LIN {X 0,Y 551.057,Z 884.33,A -85,B 0,C 180,E1 23176.84,E2 23176.84} C_VEL
LIN {X 0,Y 547.83,Z 907.139,A -85,B 0,C 180,E1 23175.833,E2 23175.833} C_VEL
LIN {X 0,Y 543.815,Z 933.396,A -85,B 0,C 180,E1 23174.47,E2 23174.47} C_VEL
LIN {X 0,Y 539.915,Z 957.037,A -85,B 0,C 180,E1 23173.041,E2 23173.041} C_VEL
LIN {X 0,Y 534.4,Z 990.703,A -85,B 0,C 180,E1 23170.731,E2 23170.731} C_VEL
LIN {X 0,Y 530.47,Z 1014.088,A -85,B 0,C 180,E1 23168.879,E2 23168.879} C_VEL
LIN {X 0,Y 527.355,Z 1031.726,A -85,B 0,C 180,E1 23167.286,E2 23167.286} C_VEL
LIN {X 0,Y 524.138,Z 1048.925,A -85,B 0,C 180,E1 23165.514,E2 23165.514} C_VEL
LIN {X 0,Y 520.353,Z 1068.496,A -85,B 0,C 180,E1 23163.207,E2 23163.207} C_VEL
LIN {X 0,Y 517.554,Z 1082.457,A -85,B 0,C 180,E1 23161.313,E2 23161.313} C_VEL
LIN {X 0,Y 514.336,Z 1098.584,A -85,B 0,C 180,E1 23158.825,E2 23158.825} C_VEL
LIN {X 0,Y 511.848,Z 1111.312,A -85,B 0,C 180,E1 23156.53,E2 23156.53} C_VEL
LIN {X 0,Y 509.597,Z 1122.961,A -85,B 0,C 180,E1 23154.088,E2 23154.088} C_VEL
LIN {X 0,Y 507.873,Z 1132.943,A -85,B 0,C 180,E1 23151.725,E2 23151.725} C_VEL
LIN {X 0,Y 506.606,Z 1141.31,A -85,B 0,C 180,E1 23149.486,E2 23149.486} C_VEL
LIN {X 0,Y 505.604,Z 1149.002,A -85,B 0,C 180,E1 23147.139,E2 23147.139} C_VEL
LIN {X 0,Y 504.896,Z 1155.619,A -85,B 0,C 180,E1 23144.803,E2 23144.803} C_VEL
LIN {X 0,Y 504.42,Z 1161.209,A -85,B 0,C 180,E1 23142.479,E2 23142.479} C_VEL
LIN {X 0,Y 504.14,Z 1166.009,A -85,B 0,C 180,E1 23140.053,E2 23140.053} C_VEL
LIN {X 0,Y 503.99,Z 1169.754,A -85,B 0,C 180,E1 23137.64,E2 23137.64} C_VEL
LIN {X 0,Y 503.929,Z 1172.474,A -85,B 0,C 180,E1 23135.238,E2 23135.238} C_VEL
LIN {X 0,Y 503.908,Z 1174.232,A -85,B 0,C 180,E1 23132.731,E2 23132.731} C_VEL
LIN {X 0,Y 503.897,Z 1174.895,A -85,B 0,C 180,E1 23130.342,E2 23130.342} C_VEL
LIN {X 0,Y 503.911,Z 1174.515,A -85,B 0,C 180,E1 23127.841,E2 23127.841} C_VEL
LIN {X 0,Y 503.919,Z 1173.138,A -85,B 0,C 180,E1 23125.449,E2 23125.449} C_VEL
LIN {X 0,Y 503.964,Z 1170.607,A -85,B 0,C 180,E1 23122.936,E2 23122.936} C_VEL
LIN {X 0,Y 504.088,Z 1167.151,A -85,B 0,C 180,E1 23120.525,E2 23120.525} C_VEL
LIN {X 0,Y 504.351,Z 1162.399,A -85,B 0,C 180,E1 23117.987,E2 23117.987} C_VEL
LIN {X 0,Y 504.788,Z 1156.758,A -85,B 0,C 180,E1 23115.549,E2 23115.549} C_VEL
LIN {X 0,Y 505.495,Z 1149.985,A -85,B 0,C 180,E1 23113.098,E2 23113.098} C_VEL
LIN {X 0,Y 506.451,Z 1142.44,A -85,B 0,C 180,E1 23110.751,E2 23110.751} C_VEL
LIN {X 0,Y 507.667,Z 1134.224,A -85,B 0,C 180,E1 23108.512,E2 23108.512} C_VEL
LIN {X 0,Y 509.239,Z 1124.921,A -85,B 0,C 180,E1 23106.266,E2 23106.266} C_VEL
LIN {X 0,Y 511.074,Z 1115.037,A -85,B 0,C 180,E1 23104.135,E2 23104.135} C_VEL
LIN {X 0,Y 512.89,Z 1105.848,A -85,B 0,C 180,E1 23102.357,E2 23102.357} C_VEL
LIN {X 0,Y 515.553,Z 1092.457,A -85,B 0,C 180,E1 23100.105,E2 23100.105} C_VEL
LIN {X 0,Y 518.946,Z 1075.502,A -85,B 0,C 180,E1 23097.615,E2 23097.615} C_VEL
LIN {X 0,Y 522.004,Z 1059.865,A -85,B 0,C 180,E1 23095.647,E2 23095.647} C_VEL
LIN {X 0,Y 524.918,Z 1044.704,A -85,B 0,C 180,E1 23093.945,E2 23093.945} C_VEL
LIN {X 0,Y 527.865,Z 1028.88,A -85,B 0,C 180,E1 23092.353,E2 23092.353} C_VEL
LIN {X 0,Y 531.711,Z 1007.061,A -85,B 0,C 180,E1 23090.445,E2 23090.445} C_VEL
LIN {X 0,Y 535.099,Z 986.395,A -85,B 0,C 180,E1 23088.874,E2 23088.874} C_VEL
LIN {X 0,Y 540.157,Z 955.538,A -85,B 0,C 180,E1 23086.774,E2 23086.774} C_VEL
LIN {X 0,Y 544.266,Z 930.729,A -85,B 0,C 180,E1 23085.284,E2 23085.284} C_VEL
LIN {X 0,Y 548.137,Z 905.022,A -85,B 0,C 180,E1 23083.979,E2 23083.979} C_VEL
LIN {X 0,Y 551.673,Z 880.009,A -85,B 0,C 180,E1 23082.891,E2 23082.891} C_VEL
LIN {X 0,Y 554.76,Z 854.396,A -85,B 0,C 180,E1 23081.983,E2 23081.983} C_VEL
LIN {X 0,Y 557.091,Z 832.3,A -85,B 0,C 180,E1 23081.336,E2 23081.336} C_VEL
LIN {X 0,Y 559.562,Z 804.066,A -85,B 0,C 180,E1 23080.685,E2 23080.685} C_VEL
LIN {X 0,Y 571.153,Z 655.622,A -85,B 0,C 180,E1 23077.83,E2 23077.83} C_VEL
LIN {X 0,Y 578.577,Z 553.045,A -85,B 0,C 180,E1 23076.025,E2 23076.025} C_VEL
LIN {X 0,Y 583.709,Z 465.889,A -85,B 0,C 180,E1 23074.614,E2 23074.614} C_VEL
LIN {X 0,Y 584.556,Z 445.741,A -85,B 0,C 180,E1 23074.283,E2 23074.283} C_VEL
LIN {X 0,Y 571.093,Z 433.147,A -85,B 0,C 180,E1 23071.921,E2 23071.921} C_VEL
LIN {X 0,Y 562.408,Z 425.648,A -85,B 0,C 180,E1 23070.267,E2 23070.267} C_VEL
LIN {X 0,Y 555.456,Z 419.784,A -85,B 0,C 180,E1 23068.845,E2 23068.845} C_VEL
LIN {X 0,Y 552.715,Z 417.682,A -85,B 0,C 180,E1 23068.24,E2 23068.24} C_VEL
LIN {X 0,Y 551.114,Z 414.287,A -85,B 0,C 180,E1 23066.566,E2 23066.566} C_VEL
LIN {X 0,Y 548.827,Z 409.657,A -85,B 0,C 180,E1 23063.743,E2 23063.743} C_VEL
LIN {X 0,Y 546.381,Z 404.793,A -85,B 0,C 180,E1 23059.221,E2 23059.221} C_VEL
LIN {X 0,Y 545.111,Z 403.52,A -85,B 0,C 180,E1 23054.663,E2 23054.663} C_VEL
LIN {X 0,Y 545.756,Z 404.238,A -85,B 0,C 180,E1 23050.557,E2 23050.557} C_VEL
LIN {X 0,Y 546.687,Z 405.294,A -85,B 0,C 180,E1 23048.52,E2 23048.52} C_VEL
LIN {X 0,Y 549.381,Z 410.452,A -85,B 0,C 180,E1 23044.07,E2 23044.07} C_VEL
LIN {X 0,Y 552.019,Z 415.595,A -85,B 0,C 180,E1 23041.098,E2 23041.098} C_VEL
LIN {X 0,Y 554.609,Z 420.558,A -85,B 0,C 180,E1 23038.76,E2 23038.76} C_VEL
LIN {X 0,Y 557.191,Z 425.708,A -85,B 0,C 180,E1 23036.708,E2 23036.708} C_VEL
LIN {X 0,Y 559.787,Z 430.872,A -85,B 0,C 180,E1 23034.876,E2 23034.876} C_VEL
LIN {X 0,Y 563.507,Z 438.145,A -85,B 0,C 180,E1 23032.557,E2 23032.557} C_VEL
LIN {X 0,Y 567.981,Z 447.698,A -85,B 0,C 180,E1 23029.963,E2 23029.963} C_VEL
LIN {X 0,Y 572.898,Z 458.394,A -85,B 0,C 180,E1 23027.399,E2 23027.399} C_VEL
LIN {X 0,Y 577.116,Z 468.188,A -85,B 0,C 180,E1 23025.322,E2 23025.322} C_VEL
LIN {X 0,Y 570.774,Z 501.691,A -85,B 0,C 180,E1 23022.354,E2 23022.354} C_VEL
LIN {X 0,Y 564.296,Z 538.268,A -85,B 0,C 180,E1 23019.244,E2 23019.244} C_VEL
LIN {X 0,Y 557.893,Z 576.998,A -85,B 0,C 180,E1 23016.066,E2 23016.066} C_VEL
LIN {X 0,Y 553.505,Z 608.409,A -85,B 0,C 180,E1 23013.5,E2 23013.5} C_VEL
LIN {X 0,Y 552.708,Z 627.613,A -85,B 0,C 180,E1 23011.761,E2 23011.761} C_VEL
LIN {X 0,Y 553.862,Z 644.721,A -85,B 0,C 180,E1 23010.056,E2 23010.056} C_VEL
LIN {X 0,Y 556.965,Z 660.711,A -85,B 0,C 180,E1 23008.311,E2 23008.311} C_VEL
LIN {X 0,Y 562.073,Z 675.706,A -85,B 0,C 180,E1 23006.532,E2 23006.532} C_VEL
LIN {X 0,Y 569.442,Z 689.793,A -85,B 0,C 180,E1 23004.711,E2 23004.711} C_VEL
LIN {X 0,Y 577.857,Z 701.318,A -85,B 0,C 180,E1 23003.099,E2 23003.099} C_VEL
LIN {X 0,Y 587.248,Z 711.274,A -85,B 0,C 180,E1 23001.613,E2 23001.613} C_VEL
LIN {X 0,Y 578.734,Z 724.816,A -85,B 0,C 180,E1 23001.262,E2 23001.262} C_VEL
LIN {X 0,Y 574.045,Z 752.67,A -85,B 0,C 180,E1 23001.309,E2 23001.309} C_VEL
LIN {X 0,Y 571.96,Z 772.656,A -85,B 0,C 180,E1 23001.194,E2 23001.194} C_VEL
LIN {X 0,Y 569.941,Z 808.835,A -85,B 0,C 180,E1 23000.623,E2 23000.623} C_VEL
LIN {X 0,Y 566.66,Z 844.611,A -85,B 0,C 180,E1 22999.922,E2 22999.922} C_VEL
LIN {X 0,Y 563.226,Z 875.195,A -85,B 0,C 180,E1 22999.144,E2 22999.144} C_VEL
LIN {X 0,Y 559.593,Z 904.524,A -85,B 0,C 180,E1 22998.204,E2 22998.204} C_VEL
LIN {X 0,Y 555.713,Z 933.276,A -85,B 0,C 180,E1 22997.078,E2 22997.078} C_VEL
LIN {X 0,Y 551.651,Z 960.721,A -85,B 0,C 180,E1 22995.793,E2 22995.793} C_VEL
LIN {X 0,Y 547.497,Z 986.268,A -85,B 0,C 180,E1 22994.382,E2 22994.382} C_VEL
LIN {X 0,Y 543.411,Z 1009.171,A -85,B 0,C 180,E1 22992.904,E2 22992.904} C_VEL
LIN {X 0,Y 539.538,Z 1029.105,A -85,B 0,C 180,E1 22991.42,E2 22991.42} C_VEL
LIN {X 0,Y 535.556,Z 1046.564,A -85,B 0,C 180,E1 22989.884,E2 22989.884} C_VEL
LIN {X 0,Y 530.767,Z 1065.297,A -85,B 0,C 180,E1 22987.955,E2 22987.955} C_VEL
LIN {X 0,Y 526.276,Z 1082.261,A -85,B 0,C 180,E1 22985.948,E2 22985.948} C_VEL
LIN {X 0,Y 521.76,Z 1099.613,A -85,B 0,C 180,E1 22983.628,E2 22983.628} C_VEL
LIN {X 0,Y 517.098,Z 1117.821,A -85,B 0,C 180,E1 22980.823,E2 22980.823} C_VEL
LIN {X 0,Y 514.09,Z 1130.733,A -85,B 0,C 180,E1 22978.583,E2 22978.583} C_VEL
LIN {X 0,Y 511.137,Z 1144.962,A -85,B 0,C 180,E1 22975.86,E2 22975.86} C_VEL
LIN {X 0,Y 508.662,Z 1158.391,A -85,B 0,C 180,E1 22972.904,E2 22972.904} C_VEL
LIN {X 0,Y 506.833,Z 1169.861,A -85,B 0,C 180,E1 22969.954,E2 22969.954} C_VEL
LIN {X 0,Y 505.513,Z 1179.907,A -85,B 0,C 180,E1 22966.902,E2 22966.902} C_VEL
LIN {X 0,Y 504.715,Z 1187.905,A -85,B 0,C 180,E1 22963.985,E2 22963.985} C_VEL
LIN {X 0,Y 504.22,Z 1194.406,A -85,B 0,C 180,E1 22961.005,E2 22961.005} C_VEL
LIN {X 0,Y 504.013,Z 1199.234,A -85,B 0,C 180,E1 22958.096,E2 22958.096} C_VEL
LIN {X 0,Y 503.931,Z 1202.607,A -85,B 0,C 180,E1 22955.235,E2 22955.235} C_VEL
LIN {X 0,Y 503.909,Z 1204.453,A -85,B 0,C 180,E1 22952.387,E2 22952.387} C_VEL
LIN {X 0,Y 503.895,Z 1204.933,A -85,B 0,C 180,E1 22949.544,E2 22949.544} C_VEL
LIN {X 0,Y 503.917,Z 1204.083,A -85,B 0,C 180,E1 22946.814,E2 22946.814} C_VEL
LIN {X 0,Y 503.943,Z 1201.768,A -85,B 0,C 180,E1 22943.962,E2 22943.962} C_VEL
LIN {X 0,Y 504.056,Z 1198.051,A -85,B 0,C 180,E1 22941.071,E2 22941.071} C_VEL
LIN {X 0,Y 504.324,Z 1192.836,A -85,B 0,C 180,E1 22938.215,E2 22938.215} C_VEL
LIN {X 0,Y 504.895,Z 1185.791,A -85,B 0,C 180,E1 22935.197,E2 22935.197} C_VEL
LIN {X 0,Y 505.81,Z 1177.429,A -85,B 0,C 180,E1 22932.275,E2 22932.275} C_VEL
LIN {X 0,Y 507.222,Z 1167.283,A -85,B 0,C 180,E1 22929.336,E2 22929.336} C_VEL
LIN {X 0,Y 509.099,Z 1155.81,A -85,B 0,C 180,E1 22926.502,E2 22926.502} C_VEL
LIN {X 0,Y 511.729,Z 1141.931,A -85,B 0,C 180,E1 22923.544,E2 22923.544} C_VEL
LIN {X 0,Y 515.165,Z 1126.235,A -85,B 0,C 180,E1 22920.589,E2 22920.589} C_VEL
LIN {X 0,Y 519.95,Z 1106.476,A -85,B 0,C 180,E1 22917.384,E2 22917.384} C_VEL
LIN {X 0,Y 524.69,Z 1088.427,A -85,B 0,C 180,E1 22914.839,E2 22914.839} C_VEL
LIN {X 0,Y 530.273,Z 1067.435,A -85,B 0,C 180,E1 22912.273,E2 22912.273} C_VEL
LIN {X 0,Y 534.945,Z 1049.198,A -85,B 0,C 180,E1 22910.362,E2 22910.362} C_VEL
LIN {X 0,Y 539.105,Z 1031.178,A -85,B 0,C 180,E1 22908.748,E2 22908.748} C_VEL
LIN {X 0,Y 543.728,Z 1007.513,A -85,B 0,C 180,E1 22906.979,E2 22906.979} C_VEL
LIN {X 0,Y 548.004,Z 983.383,A -85,B 0,C 180,E1 22905.447,E2 22905.447} C_VEL
LIN {X 0,Y 552.185,Z 957.301,A -85,B 0,C 180,E1 22904.037,E2 22904.037} C_VEL
LIN {X 0,Y 556.265,Z 929.29,A -85,B 0,C 180,E1 22902.753,E2 22902.753} C_VEL
LIN {X 0,Y 560.209,Z 899.874,A -85,B 0,C 180,E1 22901.633,E2 22901.633} C_VEL
LIN {X 0,Y 563.92,Z 869.292,A -85,B 0,C 180,E1 22900.692,E2 22900.692} C_VEL
LIN {X 0,Y 567.379,Z 837.56,A -85,B 0,C 180,E1 22899.927,E2 22899.927} C_VEL
LIN {X 0,Y 570.447,Z 801.658,A -85,B 0,C 180,E1 22899.251,E2 22899.251} C_VEL
LIN {X 0,Y 572.549,Z 755.196,A -85,B 0,C 180,E1 22898.554,E2 22898.554} C_VEL
LIN {X 0,Y 574.825,Z 710.285,A -85,B 0,C 180,E1 22897.931,E2 22897.931} C_VEL
LIN {X 0,Y 579.93,Z 660.957,A -85,B 0,C 180,E1 22897.094,E2 22897.094} C_VEL
LIN {X 0,Y 584.59,Z 616.642,A -85,B 0,C 180,E1 22896.351,E2 22896.351} C_VEL
LIN {X 0,Y 586.678,Z 598.91,A -85,B 0,C 180,E1 22896.082,E2 22896.082} C_VEL
LIN {X 0,Y 589.946,Z 567.651,A -85,B 0,C 180,E1 22895.556,E2 22895.556} C_VEL
LIN {X 0,Y 593.343,Z 541.086,A -85,B 0,C 180,E1 22895.187,E2 22895.187} C_VEL
LIN {X 0,Y 596.239,Z 512.837,A -85,B 0,C 180,E1 22894.704,E2 22894.704} C_VEL
LIN {X 0,Y 600.855,Z 478.51,A -85,B 0,C 180,E1 22894.259,E2 22894.259} C_VEL
LIN {X 0,Y 601.375,Z 470.334,A -85,B 0,C 180,E1 22894.078,E2 22894.078} C_VEL
LIN {X 0,Y 588.736,Z 449.662,A -85,B 0,C 180,E1 22891.683,E2 22891.683} C_VEL
LIN {X 0,Y 577.396,Z 432.357,A -85,B 0,C 180,E1 22889.346,E2 22889.346} C_VEL
LIN {X 0,Y 567.124,Z 417.532,A -85,B 0,C 180,E1 22887.029,E2 22887.029} C_VEL
LIN {X 0,Y 558.423,Z 405.743,A -85,B 0,C 180,E1 22884.884,E2 22884.884} C_VEL
LIN {X 0,Y 554.615,Z 400.659,A -85,B 0,C 180,E1 22883.875,E2 22883.875} C_VEL
LIN {X 0,Y 551.114,Z 396.026,A -85,B 0,C 180,E1 22882.903,E2 22882.903} C_VEL
LIN {X 0,Y 547.232,Z 391.014,A -85,B 0,C 180,E1 22881.772,E2 22881.772} C_VEL
LIN {X 0,Y 543.548,Z 386.1,A -85,B 0,C 180,E1 22880.627,E2 22880.627} C_VEL
LIN {X 0,Y 539.728,Z 381.645,A -85,B 0,C 180,E1 22879.395,E2 22879.395} C_VEL
LIN {X 0,Y 538.349,Z 379.721,A -85,B 0,C 180,E1 22878.911,E2 22878.911} C_VEL
LIN {X 0,Y 534.938,Z 375.892,A -85,B 0,C 180,E1 22877.711,E2 22877.711} C_VEL
LIN {X 0,Y 533.903,Z 374.19,A -85,B 0,C 180,E1 22877.296,E2 22877.296} C_VEL
LIN {X 0,Y 532.616,Z 376.406,A -85,B 0,C 180,E1 22877.036,E2 22877.036} C_VEL
LIN {X 0,Y 528.568,Z 388.188,A -85,B 0,C 180,E1 22876.501,E2 22876.501} C_VEL
LIN {X 0,Y 525.65,Z 395.127,A -85,B 0,C 180,E1 22875.997,E2 22875.997} C_VEL
LIN {X 0,Y 524.492,Z 397.567,A -85,B 0,C 180,E1 22875.77,E2 22875.77} C_VEL
LIN {X 0,Y 520.598,Z 409.795,A -85,B 0,C 180,E1 22875.263,E2 22875.263} C_VEL
LIN {X 0,Y 517.728,Z 417.348,A -85,B 0,C 180,E1 22874.77,E2 22874.77} C_VEL
LIN {X 0,Y 516.146,Z 420.324,A -85,B 0,C 180,E1 22874.402,E2 22874.402} C_VEL
LIN {X 0,Y 515.687,Z 512.805,A -85,B 0,C 180,E1 22870.812,E2 22870.812} C_VEL
LIN {X 0,Y 515.107,Z 590.514,A -85,B 0,C 180,E1 22867.697,E2 22867.697} C_VEL
LIN {X 0,Y 514.079,Z 669.928,A -85,B 0,C 180,E1 22864.434,E2 22864.434} C_VEL
LIN {X 0,Y 512.755,Z 750.259,A -85,B 0,C 180,E1 22861.061,E2 22861.061} C_VEL
LIN {X 0,Y 511.302,Z 830.268,A -85,B 0,C 180,E1 22857.628,E2 22857.628} C_VEL
LIN {X 0,Y 510.549,Z 854.795,A -85,B 0,C 180,E1 22856.575,E2 22856.575} C_VEL
LIN {X 0,Y 509.562,Z 867.908,A -85,B 0,C 180,E1 22856.062,E2 22856.062} C_VEL
LIN {X 0,Y 508.45,Z 974.661,A -85,B 0,C 180,E1 22854.396,E2 22854.396} C_VEL
LIN {X 0,Y 508.553,Z 991.606,A -85,B 0,C 180,E1 22854.001,E2 22854.001} C_VEL
LIN {X 0,Y 508.514,Z 1003.382,A -85,B 0,C 180,E1 22853.565,E2 22853.565} C_VEL
LIN {X 0,Y 508.365,Z 1014.88,A -85,B 0,C 180,E1 22852.996,E2 22852.996} C_VEL
LIN {X 0,Y 508.113,Z 1027.357,A -85,B 0,C 180,E1 22852.196,E2 22852.196} C_VEL
LIN {X 0,Y 507.728,Z 1039.469,A -85,B 0,C 180,E1 22851.164,E2 22851.164} C_VEL
LIN {X 0,Y 507.391,Z 1048.135,A -85,B 0,C 180,E1 22850.243,E2 22850.243} C_VEL
LIN {X 0,Y 507.039,Z 1056.133,A -85,B 0,C 180,E1 22849.202,E2 22849.202} C_VEL
LIN {X 0,Y 506.695,Z 1063.338,A -85,B 0,C 180,E1 22848.041,E2 22848.041} C_VEL
LIN {X 0,Y 506.318,Z 1070.513,A -85,B 0,C 180,E1 22846.524,E2 22846.524} C_VEL
LIN {X 0,Y 506.071,Z 1074.913,A -85,B 0,C 180,E1 22845.234,E2 22845.234} C_VEL
LIN {X 0,Y 505.886,Z 1078.023,A -85,B 0,C 180,E1 22843.936,E2 22843.936} C_VEL
LIN {X 0,Y 505.767,Z 1079.916,A -85,B 0,C 180,E1 22842.631,E2 22842.631} C_VEL
LIN {X 0,Y 505.696,Z 1080.635,A -85,B 0,C 180,E1 22841.283,E2 22841.283} C_VEL
LIN {X 0,Y 505.696,Z 1079.884,A -85,B 0,C 180,E1 22839.635,E2 22839.635} C_VEL
LIN {X 0,Y 505.751,Z 1077.275,A -85,B 0,C 180,E1 22838.058,E2 22838.058} C_VEL
LIN {X 0,Y 505.885,Z 1073.713,A -85,B 0,C 180,E1 22836.715,E2 22836.715} C_VEL
LIN {X 0,Y 506.097,Z 1068.667,A -85,B 0,C 180,E1 22835.344,E2 22835.344} C_VEL
LIN {X 0,Y 506.46,Z 1060.672,A -85,B 0,C 180,E1 22833.753,E2 22833.753} C_VEL
LIN {X 0,Y 506.791,Z 1053.188,A -85,B 0,C 180,E1 22832.605,E2 22832.605} C_VEL
LIN {X 0,Y 507.144,Z 1044.896,A -85,B 0,C 180,E1 22831.564,E2 22831.564} C_VEL
LIN {X 0,Y 507.542,Z 1035.033,A -85,B 0,C 180,E1 22830.549,E2 22830.549} C_VEL
LIN {X 0,Y 507.953,Z 1021.755,A -85,B 0,C 180,E1 22829.478,E2 22829.478} C_VEL
LIN {X 0,Y 508.244,Z 1010.502,A -85,B 0,C 180,E1 22828.775,E2 22828.775} C_VEL
LIN {X 0,Y 508.447,Z 999.419,A -85,B 0,C 180,E1 22828.23,E2 22828.23} C_VEL
LIN {X 0,Y 508.563,Z 986.604,A -85,B 0,C 180,E1 22827.756,E2 22827.756} C_VEL
LIN {X 0,Y 508.545,Z 969,A -85,B 0,C 180,E1 22827.356,E2 22827.356} C_VEL
LIN {X 0,Y 509.787,Z 859.318,A -85,B 0,C 180,E1 22825.674,E2 22825.674} C_VEL
LIN {X 0,Y 510.753,Z 842.929,A -85,B 0,C 180,E1 22824.955,E2 22824.955} C_VEL
LIN {X 0,Y 511.075,Z 831.021,A -85,B 0,C 180,E1 22824.399,E2 22824.399} C_VEL
LIN {X 0,Y 512.025,Z 832.145,A -85,B 0,C 180,E1 22824.206,E2 22824.206} C_VEL
LIN {X 0,Y 513.762,Z 831.805,A -85,B 0,C 180,E1 22823.967,E2 22823.967} C_VEL
LIN {X 0,Y 516.668,Z 828.931,A -85,B 0,C 180,E1 22823.67,E2 22823.67} C_VEL
LIN {X 0,Y 520.436,Z 823.214,A -85,B 0,C 180,E1 22823.377,E2 22823.377} C_VEL
LIN {X 0,Y 523.679,Z 821.557,A -85,B 0,C 180,E1 22822.992,E2 22822.992} C_VEL
LIN {X 0,Y 527.493,Z 817.574,A -85,B 0,C 180,E1 22822.623,E2 22822.623} C_VEL
LIN {X 0,Y 530.622,Z 812.978,A -85,B 0,C 180,E1 22822.371,E2 22822.371} C_VEL
LIN {X 0,Y 534.974,Z 809.845,A -85,B 0,C 180,E1 22821.918,E2 22821.918} C_VEL
LIN {X 0,Y 539.645,Z 804.391,A -85,B 0,C 180,E1 22821.513,E2 22821.513} C_VEL
LIN {X 0,Y 541.355,Z 802.215,A -85,B 0,C 180,E1 22821.37,E2 22821.37} C_VEL
LIN {X 0,Y 546.443,Z 798.034,A -85,B 0,C 180,E1 22820.885,E2 22820.885} C_VEL
LIN {X 0,Y 552.264,Z 791.252,A -85,B 0,C 180,E1 22820.408,E2 22820.408} C_VEL
LIN {X 0,Y 558.072,Z 786.124,A -85,B 0,C 180,E1 22819.901,E2 22819.901} C_VEL
LIN {X 0,Y 561.235,Z 782.605,A -85,B 0,C 180,E1 22819.648,E2 22819.648} C_VEL
LIN {X 0,Y 557.807,Z 825.252,A -85,B 0,C 180,E1 22818.76,E2 22818.76} C_VEL
LIN {X 0,Y 555.053,Z 851.798,A -85,B 0,C 180,E1 22818.011,E2 22818.011} C_VEL
LIN {X 0,Y 552.428,Z 873.748,A -85,B 0,C 180,E1 22817.254,E2 22817.254} C_VEL
LIN {X 0,Y 551.057,Z 884.33,A -85,B 0,C 180,E1 22816.84,E2 22816.84} C_VEL
LIN {X 0,Y 549.33,Z 891.609,A -85,B 0,C 180,E1 22816.608,E2 22816.608} C_VEL
LIN {X 0,Y 542.253,Z 910.012,A -85,B 0,C 180,E1 22816.209,E2 22816.209} C_VEL
LIN {X 0,Y 540.387,Z 917.023,A -85,B 0,C 180,E1 22815.923,E2 22815.923} C_VEL
LIN {X 0,Y 536.495,Z 940.102,A -85,B 0,C 180,E1 22814.64,E2 22814.64} C_VEL
LIN {X 0,Y 532.171,Z 964.685,A -85,B 0,C 180,E1 22813.075,E2 22813.075} C_VEL
LIN {X 0,Y 527.582,Z 989.152,A -85,B 0,C 180,E1 22811.266,E2 22811.266} C_VEL
LIN {X 0,Y 522.647,Z 1016.661,A -85,B 0,C 180,E1 22809.008,E2 22809.008} C_VEL
LIN {X 0,Y 519.475,Z 1034.198,A -85,B 0,C 180,E1 22807.387,E2 22807.387} C_VEL
LIN {X 0,Y 515.717,Z 1054.189,A -85,B 0,C 180,E1 22805.288,E2 22805.288} C_VEL
LIN {X 0,Y 512.383,Z 1070.744,A -85,B 0,C 180,E1 22803.255,E2 22803.255} C_VEL
LIN {X 0,Y 509.683,Z 1084.106,A -85,B 0,C 180,E1 22801.419,E2 22801.419} C_VEL
LIN {X 0,Y 507.508,Z 1094.866,A -85,B 0,C 180,E1 22799.769,E2 22799.769} C_VEL
LIN {X 0,Y 504.71,Z 1108.752,A -85,B 0,C 180,E1 22797.364,E2 22797.364} C_VEL
LIN {X 0,Y 502.082,Z 1122.433,A -85,B 0,C 180,E1 22794.597,E2 22794.597} C_VEL
LIN {X 0,Y 500.238,Z 1132.482,A -85,B 0,C 180,E1 22792.197,E2 22792.197} C_VEL
LIN {X 0,Y 498.795,Z 1141.311,A -85,B 0,C 180,E1 22789.804,E2 22789.804} C_VEL
LIN {X 0,Y 497.717,Z 1149.068,A -85,B 0,C 180,E1 22787.397,E2 22787.397} C_VEL
LIN {X 0,Y 496.976,Z 1155.625,A -85,B 0,C 180,E1 22785.041,E2 22785.041} C_VEL
LIN {X 0,Y 496.463,Z 1161.208,A -85,B 0,C 180,E1 22782.683,E2 22782.683} C_VEL
LIN {X 0,Y 496.16,Z 1166.007,A -85,B 0,C 180,E1 22780.216,E2 22780.216} C_VEL
LIN {X 0,Y 495.997,Z 1169.752,A -85,B 0,C 180,E1 22777.764,E2 22777.764} C_VEL
LIN {X 0,Y 495.931,Z 1172.471,A -85,B 0,C 180,E1 22775.323,E2 22775.323} C_VEL
LIN {X 0,Y 495.911,Z 1174.181,A -85,B 0,C 180,E1 22772.891,E2 22772.891} C_VEL
LIN {X 0,Y 495.897,Z 1174.892,A -85,B 0,C 180,E1 22770.348,E2 22770.348} C_VEL
LIN {X 0,Y 495.91,Z 1174.512,A -85,B 0,C 180,E1 22767.806,E2 22767.806} C_VEL
LIN {X 0,Y 495.919,Z 1173.135,A -85,B 0,C 180,E1 22765.376,E2 22765.376} C_VEL
LIN {X 0,Y 495.965,Z 1170.751,A -85,B 0,C 180,E1 22762.937,E2 22762.937} C_VEL
LIN {X 0,Y 496.094,Z 1167.344,A -85,B 0,C 180,E1 22760.488,E2 22760.488} C_VEL
LIN {X 0,Y 496.369,Z 1162.642,A -85,B 0,C 180,E1 22757.909,E2 22757.909} C_VEL
LIN {X 0,Y 496.828,Z 1157.052,A -85,B 0,C 180,E1 22755.431,E2 22755.431} C_VEL
LIN {X 0,Y 497.569,Z 1150.335,A -85,B 0,C 180,E1 22752.94,E2 22752.94} C_VEL
LIN {X 0,Y 498.576,Z 1142.843,A -85,B 0,C 180,E1 22750.556,E2 22750.556} C_VEL
LIN {X 0,Y 499.933,Z 1134.221,A -85,B 0,C 180,E1 22748.162,E2 22748.162} C_VEL
LIN {X 0,Y 501.599,Z 1124.918,A -85,B 0,C 180,E1 22745.882,E2 22745.882} C_VEL
LIN {X 0,Y 503.359,Z 1115.588,A -85,B 0,C 180,E1 22743.88,E2 22743.88} C_VEL
LIN {X 0,Y 505.822,Z 1103.237,A -85,B 0,C 180,E1 22741.552,E2 22741.552} C_VEL
LIN {X 0,Y 508.943,Z 1087.765,A -85,B 0,C 180,E1 22739.022,E2 22739.022} C_VEL
LIN {X 0,Y 511.971,Z 1072.729,A -85,B 0,C 180,E1 22736.914,E2 22736.914} C_VEL
LIN {X 0,Y 514.954,Z 1057.848,A -85,B 0,C 180,E1 22735.056,E2 22735.056} C_VEL
LIN {X 0,Y 517.748,Z 1043.417,A -85,B 0,C 180,E1 22733.456,E2 22733.456} C_VEL
LIN {X 0,Y 521.672,Z 1022.322,A -85,B 0,C 180,E1 22731.402,E2 22731.402} C_VEL
LIN {X 0,Y 525.261,Z 1001.87,A -85,B 0,C 180,E1 22729.67,E2 22729.67} C_VEL
LIN {X 0,Y 530.118,Z 975.404,A -85,B 0,C 180,E1 22727.603,E2 22727.603} C_VEL
LIN {X 0,Y 534.201,Z 953.118,A -85,B 0,C 180,E1 22726.073,E2 22726.073} C_VEL
LIN {X 0,Y 538.645,Z 927.352,A -85,B 0,C 180,E1 22724.538,E2 22724.538} C_VEL
LIN {X 0,Y 542.182,Z 905.1,A -85,B 0,C 180,E1 22723.4,E2 22723.4} C_VEL
LIN {X 0,Y 545.949,Z 879.432,A -85,B 0,C 180,E1 22722.279,E2 22722.279} C_VEL
LIN {X 0,Y 549.003,Z 855.126,A -85,B 0,C 180,E1 22721.41,E2 22721.41} C_VEL
LIN {X 0,Y 551.527,Z 832.12,A -85,B 0,C 180,E1 22720.731,E2 22720.731} C_VEL
LIN {X 0,Y 554.534,Z 798.241,A -85,B 0,C 180,E1 22719.967,E2 22719.967} C_VEL
LIN {X 0,Y 565.722,Z 662.457,A -85,B 0,C 180,E1 22717.314,E2 22717.314} C_VEL
LIN {X 0,Y 573.294,Z 562.643,A -85,B 0,C 180,E1 22715.534,E2 22715.534} C_VEL
LIN {X 0,Y 578.714,Z 475.813,A -85,B 0,C 180,E1 22714.11,E2 22714.11} C_VEL
LIN {X 0,Y 579.94,Z 451.151,A -85,B 0,C 180,E1 22713.723,E2 22713.723} C_VEL
LIN {X 0,Y 568.745,Z 440.512,A -85,B 0,C 180,E1 22711.713,E2 22711.713} C_VEL
LIN {X 0,Y 559.89,Z 432.851,A -85,B 0,C 180,E1 22710.003,E2 22710.003} C_VEL
LIN {X 0,Y 553.218,Z 427.194,A -85,B 0,C 180,E1 22708.618,E2 22708.618} C_VEL
LIN {X 0,Y 547.525,Z 422.616,A -85,B 0,C 180,E1 22707.341,E2 22707.341} C_VEL
LIN {X 0,Y 546.765,Z 420.976,A -85,B 0,C 180,E1 22706.501,E2 22706.501} C_VEL
LIN {X 0,Y 544.443,Z 416.306,A -85,B 0,C 180,E1 22703.595,E2 22703.595} C_VEL
LIN {X 0,Y 542.146,Z 411.577,A -85,B 0,C 180,E1 22699.165,E2 22699.165} C_VEL
LIN {X 0,Y 540.915,Z 410.336,A -85,B 0,C 180,E1 22694.56,E2 22694.56} C_VEL
LIN {X 0,Y 541.573,Z 411.062,A -85,B 0,C 180,E1 22690.532,E2 22690.532} C_VEL
LIN {X 0,Y 542.477,Z 412.183,A -85,B 0,C 180,E1 22688.48,E2 22688.48} C_VEL
LIN {X 0,Y 545.095,Z 417.253,A -85,B 0,C 180,E1 22684.102,E2 22684.102} C_VEL
LIN {X 0,Y 547.666,Z 422.332,A -85,B 0,C 180,E1 22681.151,E2 22681.151} C_VEL
LIN {X 0,Y 550.166,Z 427.162,A -85,B 0,C 180,E1 22678.854,E2 22678.854} C_VEL
LIN {X 0,Y 552.713,Z 432.322,A -85,B 0,C 180,E1 22676.785,E2 22676.785} C_VEL
LIN {X 0,Y 555.138,Z 437.189,A -85,B 0,C 180,E1 22675.04,E2 22675.04} C_VEL
LIN {X 0,Y 558.944,Z 444.834,A -85,B 0,C 180,E1 22672.6,E2 22672.6} C_VEL
LIN {X 0,Y 563.21,Z 454.023,A -85,B 0,C 180,E1 22670.084,E2 22670.084} C_VEL
LIN {X 0,Y 568.056,Z 464.757,A -85,B 0,C 180,E1 22667.496,E2 22667.496} C_VEL
LIN {X 0,Y 571.656,Z 473.135,A -85,B 0,C 180,E1 22665.69,E2 22665.69} C_VEL
LIN {X 0,Y 565.074,Z 506.643,A -85,B 0,C 180,E1 22662.706,E2 22662.706} C_VEL
LIN {X 0,Y 558.317,Z 543.422,A -85,B 0,C 180,E1 22659.56,E2 22659.56} C_VEL
LIN {X 0,Y 551.589,Z 582.652,A -85,B 0,C 180,E1 22656.321,E2 22656.321} C_VEL
LIN {X 0,Y 547.378,Z 612.144,A -85,B 0,C 180,E1 22653.881,E2 22653.881} C_VEL
LIN {X 0,Y 546.514,Z 631.843,A -85,B 0,C 180,E1 22652.071,E2 22652.071} C_VEL
LIN {X 0,Y 547.693,Z 649.461,A -85,B 0,C 180,E1 22650.286,E2 22650.286} C_VEL
LIN {X 0,Y 550.631,Z 664.816,A -85,B 0,C 180,E1 22648.587,E2 22648.587} C_VEL
LIN {X 0,Y 555.51,Z 679.592,A -85,B 0,C 180,E1 22646.818,E2 22646.818} C_VEL
LIN {X 0,Y 562.696,Z 693.778,A -85,B 0,C 180,E1 22644.973,E2 22644.973} C_VEL
LIN {X 0,Y 571.044,Z 705.609,A -85,B 0,C 180,E1 22643.314,E2 22643.314} C_VEL
LIN {X 0,Y 578.661,Z 714.131,A -85,B 0,C 180,E1 22642.047,E2 22642.047} C_VEL
LIN {X 0,Y 574.416,Z 721.089,A -85,B 0,C 180,E1 22641.871,E2 22641.871} C_VEL
LIN {X 0,Y 569.292,Z 750.88,A -85,B 0,C 180,E1 22641.942,E2 22641.942} C_VEL
LIN {X 0,Y 566.976,Z 772.153,A -85,B 0,C 180,E1 22641.827,E2 22641.827} C_VEL
LIN {X 0,Y 564.818,Z 807.679,A -85,B 0,C 180,E1 22641.26,E2 22641.26} C_VEL
LIN {X 0,Y 561.44,Z 843.12,A -85,B 0,C 180,E1 22640.56,E2 22640.56} C_VEL
LIN {X 0,Y 557.742,Z 874.698,A -85,B 0,C 180,E1 22639.755,E2 22639.755} C_VEL
LIN {X 0,Y 553.816,Z 904.922,A -85,B 0,C 180,E1 22638.777,E2 22638.777} C_VEL
LIN {X 0,Y 549.847,Z 933.184,A -85,B 0,C 180,E1 22637.662,E2 22637.662} C_VEL
LIN {X 0,Y 545.651,Z 960.689,A -85,B 0,C 180,E1 22636.368,E2 22636.368} C_VEL
LIN {X 0,Y 541.197,Z 987.411,A -85,B 0,C 180,E1 22634.889,E2 22634.889} C_VEL
LIN {X 0,Y 536.696,Z 1012.133,A -85,B 0,C 180,E1 22633.28,E2 22633.28} C_VEL
LIN {X 0,Y 532.373,Z 1033.977,A -85,B 0,C 180,E1 22631.624,E2 22631.624} C_VEL
LIN {X 0,Y 528.219,Z 1052.487,A -85,B 0,C 180,E1 22629.98,E2 22629.98} C_VEL
LIN {X 0,Y 524.263,Z 1067.785,A -85,B 0,C 180,E1 22628.383,E2 22628.383} C_VEL
LIN {X 0,Y 519.408,Z 1084.935,A -85,B 0,C 180,E1 22626.293,E2 22626.293} C_VEL
LIN {X 0,Y 514.302,Z 1102.883,A -85,B 0,C 180,E1 22623.78,E2 22623.78} C_VEL
LIN {X 0,Y 509.846,Z 1119.215,A -85,B 0,C 180,E1 22621.179,E2 22621.179} C_VEL
LIN {X 0,Y 505.312,Z 1137.654,A -85,B 0,C 180,E1 22617.809,E2 22617.809} C_VEL
LIN {X 0,Y 502.164,Z 1152.253,A -85,B 0,C 180,E1 22614.716,E2 22614.716} C_VEL
LIN {X 0,Y 499.809,Z 1165.06,A -85,B 0,C 180,E1 22611.597,E2 22611.597} C_VEL
LIN {X 0,Y 498.215,Z 1175.503,A -85,B 0,C 180,E1 22608.607,E2 22608.607} C_VEL
LIN {X 0,Y 497.07,Z 1184.873,A -85,B 0,C 180,E1 22605.397,E2 22605.397} C_VEL
LIN {X 0,Y 496.421,Z 1191.91,A -85,B 0,C 180,E1 22602.444,E2 22602.444} C_VEL
LIN {X 0,Y 496.097,Z 1197.318,A -85,B 0,C 180,E1 22599.511,E2 22599.511} C_VEL
LIN {X 0,Y 495.958,Z 1201.399,A -85,B 0,C 180,E1 22596.481,E2 22596.481} C_VEL
LIN {X 0,Y 495.915,Z 1203.92,A -85,B 0,C 180,E1 22593.578,E2 22593.578} C_VEL
LIN {X 0,Y 495.901,Z 1204.881,A -85,B 0,C 180,E1 22590.807,E2 22590.807} C_VEL
LIN {X 0,Y 495.91,Z 1204.609,A -85,B 0,C 180,E1 22587.919,E2 22587.919} C_VEL
LIN {X 0,Y 495.925,Z 1202.962,A -85,B 0,C 180,E1 22585.141,E2 22585.141} C_VEL
LIN {X 0,Y 496.003,Z 1199.708,A -85,B 0,C 180,E1 22582.12,E2 22582.12} C_VEL
LIN {X 0,Y 496.21,Z 1195.149,A -85,B 0,C 180,E1 22579.198,E2 22579.198} C_VEL
LIN {X 0,Y 496.698,Z 1188.706,A -85,B 0,C 180,E1 22576.138,E2 22576.138} C_VEL
LIN {X 0,Y 497.549,Z 1180.587,A -85,B 0,C 180,E1 22573.056,E2 22573.056} C_VEL
LIN {X 0,Y 498.861,Z 1171.069,A -85,B 0,C 180,E1 22570.059,E2 22570.059} C_VEL
LIN {X 0,Y 500.793,Z 1159.519,A -85,B 0,C 180,E1 22566.991,E2 22566.991} C_VEL
LIN {X 0,Y 503.909,Z 1144.022,A -85,B 0,C 180,E1 22563.482,E2 22563.482} C_VEL
LIN {X 0,Y 507.439,Z 1128.608,A -85,B 0,C 180,E1 22560.486,E2 22560.486} C_VEL
LIN {X 0,Y 511.802,Z 1112.097,A -85,B 0,C 180,E1 22557.634,E2 22557.634} C_VEL
LIN {X 0,Y 517.571,Z 1091.525,A -85,B 0,C 180,E1 22554.579,E2 22554.579} C_VEL
LIN {X 0,Y 522.614,Z 1073.804,A -85,B 0,C 180,E1 22552.317,E2 22552.317} C_VEL
LIN {X 0,Y 527.254,Z 1056.493,A -85,B 0,C 180,E1 22550.416,E2 22550.416} C_VEL
LIN {X 0,Y 531.233,Z 1039.568,A -85,B 0,C 180,E1 22548.841,E2 22548.841} C_VEL
LIN {X 0,Y 535.026,Z 1020.78,A -85,B 0,C 180,E1 22547.353,E2 22547.353} C_VEL
LIN {X 0,Y 538.603,Z 1001.801,A -85,B 0,C 180,E1 22546.027,E2 22546.027} C_VEL
LIN {X 0,Y 542.679,Z 978.838,A -85,B 0,C 180,E1 22544.614,E2 22544.614} C_VEL
LIN {X 0,Y 546.923,Z 952.658,A -85,B 0,C 180,E1 22543.235,E2 22543.235} C_VEL
LIN {X 0,Y 551.105,Z 924.513,A -85,B 0,C 180,E1 22541.975,E2 22541.975} C_VEL
LIN {X 0,Y 555.219,Z 894.341,A -85,B 0,C 180,E1 22540.858,E2 22540.858} C_VEL
LIN {X 0,Y 559.125,Z 862.981,A -85,B 0,C 180,E1 22539.924,E2 22539.924} C_VEL
LIN {X 0,Y 562.849,Z 829.791,A -85,B 0,C 180,E1 22539.16,E2 22539.16} C_VEL
LIN {X 0,Y 565.714,Z 794.681,A -85,B 0,C 180,E1 22538.514,E2 22538.514} C_VEL
LIN {X 0,Y 568.139,Z 742.839,A -85,B 0,C 180,E1 22537.757,E2 22537.757} C_VEL
LIN {X 0,Y 570.157,Z 706.195,A -85,B 0,C 180,E1 22537.247,E2 22537.247} C_VEL
LIN {X 0,Y 574.653,Z 663.027,A -85,B 0,C 180,E1 22536.507,E2 22536.507} C_VEL
LIN {X 0,Y 579.733,Z 615.937,A -85,B 0,C 180,E1 22535.721,E2 22535.721} C_VEL
LIN {X 0,Y 581.703,Z 599.345,A -85,B 0,C 180,E1 22535.467,E2 22535.467} C_VEL
LIN {X 0,Y 585.076,Z 567.755,A -85,B 0,C 180,E1 22534.936,E2 22534.936} C_VEL
LIN {X 0,Y 588.456,Z 541.617,A -85,B 0,C 180,E1 22534.574,E2 22534.574} C_VEL
LIN {X 0,Y 591.443,Z 513.111,A -85,B 0,C 180,E1 22534.087,E2 22534.087} C_VEL
LIN {X 0,Y 596.065,Z 479.079,A -85,B 0,C 180,E1 22533.647,E2 22533.647} C_VEL
LIN {X 0,Y 596.32,Z 474.509,A -85,B 0,C 180,E1 22533.539,E2 22533.539} C_VEL
LIN {X 0,Y 584.759,Z 455.455,A -85,B 0,C 180,E1 22531.291,E2 22531.291} C_VEL
LIN {X 0,Y 573.872,Z 438.688,A -85,B 0,C 180,E1 22528.997,E2 22528.997} C_VEL
LIN {X 0,Y 563.942,Z 424.198,A -85,B 0,C 180,E1 22526.71,E2 22526.71} C_VEL
LIN {X 0,Y 555.36,Z 412.416,A -85,B 0,C 180,E1 22524.548,E2 22524.548} C_VEL
LIN {X 0,Y 548.937,Z 403.683,A -85,B 0,C 180,E1 22522.772,E2 22522.772} C_VEL
LIN {X 0,Y 544.407,Z 397.936,A -85,B 0,C 180,E1 22521.438,E2 22521.438} C_VEL
LIN {X 0,Y 540.29,Z 392.617,A -85,B 0,C 180,E1 22520.134,E2 22520.134} C_VEL
LIN {X 0,Y 536.713,Z 387.865,A -85,B 0,C 180,E1 22518.915,E2 22518.915} C_VEL
LIN {X 0,Y 533.039,Z 383.977,A -85,B 0,C 180,E1 22517.628,E2 22517.628} C_VEL
LIN {X 0,Y 529.068,Z 394.782,A -85,B 0,C 180,E1 22517.076,E2 22517.076} C_VEL
LIN {X 0,Y 525.726,Z 402.368,A -85,B 0,C 180,E1 22516.496,E2 22516.496} C_VEL
LIN {X 0,Y 521.634,Z 414.756,A -85,B 0,C 180,E1 22515.959,E2 22515.959} C_VEL
LIN {X 0,Y 518.483,Z 422.726,A -85,B 0,C 180,E1 22515.42,E2 22515.42} C_VEL
LIN {X 0,Y 516.946,Z 426.077,A -85,B 0,C 180,E1 22515.111,E2 22515.111} C_VEL
LIN {X 0,Y 512.953,Z 438.812,A -85,B 0,C 180,E1 22514.571,E2 22514.571} C_VEL
LIN {X 0,Y 510.079,Z 446.493,A -85,B 0,C 180,E1 22514.054,E2 22514.054} C_VEL
LIN {X 0,Y 508.624,Z 449.604,A -85,B 0,C 180,E1 22513.688,E2 22513.688} C_VEL
LIN {X 0,Y 508.24,Z 534.787,A -85,B 0,C 180,E1 22510.313,E2 22510.313} C_VEL
LIN {X 0,Y 507.467,Z 606.68,A -85,B 0,C 180,E1 22507.387,E2 22507.387} C_VEL
LIN {X 0,Y 506.651,Z 664.609,A -85,B 0,C 180,E1 22504.982,E2 22504.982} C_VEL
LIN {X 0,Y 505.393,Z 739.937,A -85,B 0,C 180,E1 22501.814,E2 22501.814} C_VEL
LIN {X 0,Y 503.894,Z 819.05,A -85,B 0,C 180,E1 22498.408,E2 22498.408} C_VEL
LIN {X 0,Y 502.996,Z 854.351,A -85,B 0,C 180,E1 22496.883,E2 22496.883} C_VEL
LIN {X 0,Y 501.85,Z 869.193,A -85,B 0,C 180,E1 22496.291,E2 22496.291} C_VEL
LIN {X 0,Y 500.65,Z 973.692,A -85,B 0,C 180,E1 22494.62,E2 22494.62} C_VEL
LIN {X 0,Y 500.787,Z 990.651,A -85,B 0,C 180,E1 22494.256,E2 22494.256} C_VEL
LIN {X 0,Y 500.735,Z 1004.336,A -85,B 0,C 180,E1 22493.752,E2 22493.752} C_VEL
LIN {X 0,Y 500.58,Z 1015.892,A -85,B 0,C 180,E1 22493.174,E2 22493.174} C_VEL
LIN {X 0,Y 500.328,Z 1027.678,A -85,B 0,C 180,E1 22492.414,E2 22492.414} C_VEL
LIN {X 0,Y 499.942,Z 1040.003,A -85,B 0,C 180,E1 22491.373,E2 22491.373} C_VEL
LIN {X 0,Y 499.585,Z 1048.777,A -85,B 0,C 180,E1 22490.438,E2 22490.438} C_VEL
LIN {X 0,Y 499.21,Z 1056.865,A -85,B 0,C 180,E1 22489.381,E2 22489.381} C_VEL
LIN {X 0,Y 498.877,Z 1063.473,A -85,B 0,C 180,E1 22488.321,E2 22488.321} C_VEL
LIN {X 0,Y 498.529,Z 1069.946,A -85,B 0,C 180,E1 22487.018,E2 22487.018} C_VEL
LIN {X 0,Y 498.204,Z 1075.578,A -85,B 0,C 180,E1 22485.471,E2 22485.471} C_VEL
LIN {X 0,Y 497.983,Z 1079.056,A -85,B 0,C 180,E1 22484.033,E2 22484.033} C_VEL
LIN {X 0,Y 497.852,Z 1080.986,A -85,B 0,C 180,E1 22482.708,E2 22482.708} C_VEL
LIN {X 0,Y 497.775,Z 1081.73,A -85,B 0,C 180,E1 22481.374,E2 22481.374} C_VEL
LIN {X 0,Y 497.766,Z 1081.132,A -85,B 0,C 180,E1 22479.787,E2 22479.787} C_VEL
LIN {X 0,Y 497.83,Z 1078.454,A -85,B 0,C 180,E1 22478.063,E2 22478.063} C_VEL
LIN {X 0,Y 497.968,Z 1074.908,A -85,B 0,C 180,E1 22476.699,E2 22476.699} C_VEL
LIN {X 0,Y 498.181,Z 1069.939,A -85,B 0,C 180,E1 22475.325,E2 22475.325} C_VEL
LIN {X 0,Y 498.536,Z 1062.663,A -85,B 0,C 180,E1 22473.817,E2 22473.817} C_VEL
LIN {X 0,Y 498.918,Z 1054.169,A -85,B 0,C 180,E1 22472.487,E2 22472.487} C_VEL
LIN {X 0,Y 499.297,Z 1045.625,A -85,B 0,C 180,E1 22471.405,E2 22471.405} C_VEL
LIN {X 0,Y 499.766,Z 1034.396,A -85,B 0,C 180,E1 22470.252,E2 22470.252} C_VEL
LIN {X 0,Y 500.141,Z 1022.091,A -85,B 0,C 180,E1 22469.28,E2 22469.28} C_VEL
LIN {X 0,Y 500.447,Z 1010.489,A -85,B 0,C 180,E1 22468.556,E2 22468.556} C_VEL
LIN {X 0,Y 500.667,Z 998.228,A -85,B 0,C 180,E1 22467.963,E2 22467.963} C_VEL
LIN {X 0,Y 500.763,Z 981.997,A -85,B 0,C 180,E1 22467.422,E2 22467.422} C_VEL
LIN {X 0,Y 500.707,Z 965.414,A -85,B 0,C 180,E1 22467.102,E2 22467.102} C_VEL
LIN {X 0,Y 502.051,Z 860.164,A -85,B 0,C 180,E1 22465.451,E2 22465.451} C_VEL
LIN {X 0,Y 503.006,Z 847.271,A -85,B 0,C 180,E1 22464.874,E2 22464.874} C_VEL
LIN {X 0,Y 503.704,Z 848.179,A -85,B 0,C 180,E1 22464.714,E2 22464.714} C_VEL
LIN {X 0,Y 505.523,Z 847.991,A -85,B 0,C 180,E1 22464.443,E2 22464.443} C_VEL
LIN {X 0,Y 508.435,Z 845.388,A -85,B 0,C 180,E1 22464.138,E2 22464.138} C_VEL
LIN {X 0,Y 512.035,Z 839.904,A -85,B 0,C 180,E1 22463.861,E2 22463.861} C_VEL
LIN {X 0,Y 515.433,Z 838.203,A -85,B 0,C 180,E1 22463.448,E2 22463.448} C_VEL
LIN {X 0,Y 519.286,Z 834.248,A -85,B 0,C 180,E1 22463.076,E2 22463.076} C_VEL
LIN {X 0,Y 522.262,Z 829.993,A -85,B 0,C 180,E1 22462.84,E2 22462.84} C_VEL
LIN {X 0,Y 526.612,Z 826.923,A -85,B 0,C 180,E1 22462.378,E2 22462.378} C_VEL
LIN {X 0,Y 531.123,Z 821.804,A -85,B 0,C 180,E1 22461.986,E2 22461.986} C_VEL
LIN {X 0,Y 533.104,Z 819.232,A -85,B 0,C 180,E1 22461.829,E2 22461.829} C_VEL
LIN {X 0,Y 538.191,Z 815.056,A -85,B 0,C 180,E1 22461.339,E2 22461.339} C_VEL
LIN {X 0,Y 543.84,Z 808.432,A -85,B 0,C 180,E1 22460.869,E2 22460.869} C_VEL
LIN {X 0,Y 549.603,Z 803.405,A -85,B 0,C 180,E1 22460.348,E2 22460.348} C_VEL
LIN {X 0,Y 554.559,Z 797.635,A -85,B 0,C 180,E1 22459.957,E2 22459.957} C_VEL
LIN {X 0,Y 551.522,Z 832.109,A -85,B 0,C 180,E1 22459.179,E2 22459.179} C_VEL
LIN {X 0,Y 548.929,Z 855.599,A -85,B 0,C 180,E1 22458.484,E2 22458.484} C_VEL
LIN {X 0,Y 545.704,Z 881.299,A -85,B 0,C 180,E1 22457.559,E2 22457.559} C_VEL
LIN {X 0,Y 542.035,Z 906.02,A -85,B 0,C 180,E1 22456.467,E2 22456.467} C_VEL
LIN {X 0,Y 540.387,Z 917.023,A -85,B 0,C 180,E1 22455.923,E2 22455.923} C_VEL
LIN {X 0,Y 538.469,Z 924.142,A -85,B 0,C 180,E1 22455.618,E2 22455.618} C_VEL
LIN {X 0,Y 530.479,Z 942.924,A -85,B 0,C 180,E1 22455.002,E2 22455.002} C_VEL
LIN {X 0,Y 528.877,Z 948.63,A -85,B 0,C 180,E1 22454.707,E2 22454.707} C_VEL
LIN {X 0,Y 524.242,Z 972.619,A -85,B 0,C 180,E1 22453.065,E2 22453.065} C_VEL
LIN {X 0,Y 519.722,Z 995.383,A -85,B 0,C 180,E1 22451.293,E2 22451.293} C_VEL
LIN {X 0,Y 515.03,Z 1018.533,A -85,B 0,C 180,E1 22449.228,E2 22449.228} C_VEL
LIN {X 0,Y 510.243,Z 1043.579,A -85,B 0,C 180,E1 22446.776,E2 22446.776} C_VEL
LIN {X 0,Y 507.148,Z 1059.353,A -85,B 0,C 180,E1 22445.012,E2 22445.012} C_VEL
LIN {X 0,Y 504.41,Z 1073.001,A -85,B 0,C 180,E1 22443.306,E2 22443.306} C_VEL
LIN {X 0,Y 501.292,Z 1088.108,A -85,B 0,C 180,E1 22441.163,E2 22441.163} C_VEL
LIN {X 0,Y 498.037,Z 1104.099,A -85,B 0,C 180,E1 22438.544,E2 22438.544} C_VEL
LIN {X 0,Y 495.681,Z 1115.653,A -85,B 0,C 180,E1 22436.347,E2 22436.347} C_VEL
LIN {X 0,Y 493.603,Z 1126.518,A -85,B 0,C 180,E1 22433.993,E2 22433.993} C_VEL
LIN {X 0,Y 491.593,Z 1138.04,A -85,B 0,C 180,E1 22431.102,E2 22431.102} C_VEL
LIN {X 0,Y 489.959,Z 1148.299,A -85,B 0,C 180,E1 22427.949,E2 22427.949} C_VEL
LIN {X 0,Y 489.102,Z 1155.316,A -85,B 0,C 180,E1 22425.414,E2 22425.414} C_VEL
LIN {X 0,Y 488.511,Z 1161.206,A -85,B 0,C 180,E1 22422.893,E2 22422.893} C_VEL
LIN {X 0,Y 488.183,Z 1166.005,A -85,B 0,C 180,E1 22420.385,E2 22420.385} C_VEL
LIN {X 0,Y 488.009,Z 1169.751,A -85,B 0,C 180,E1 22417.892,E2 22417.892} C_VEL
LIN {X 0,Y 487.932,Z 1172.469,A -85,B 0,C 180,E1 22415.41,E2 22415.41} C_VEL
LIN {X 0,Y 487.911,Z 1174.178,A -85,B 0,C 180,E1 22412.938,E2 22412.938} C_VEL
LIN {X 0,Y 487.897,Z 1174.889,A -85,B 0,C 180,E1 22410.354,E2 22410.354} C_VEL
LIN {X 0,Y 487.911,Z 1174.557,A -85,B 0,C 180,E1 22407.887,E2 22407.887} C_VEL
LIN {X 0,Y 487.919,Z 1173.131,A -85,B 0,C 180,E1 22405.3,E2 22405.3} C_VEL
LIN {X 0,Y 487.974,Z 1170.747,A -85,B 0,C 180,E1 22402.821,E2 22402.821} C_VEL
LIN {X 0,Y 488.108,Z 1167.34,A -85,B 0,C 180,E1 22400.331,E2 22400.331} C_VEL
LIN {X 0,Y 488.402,Z 1162.637,A -85,B 0,C 180,E1 22397.708,E2 22397.708} C_VEL
LIN {X 0,Y 488.898,Z 1157.047,A -85,B 0,C 180,E1 22395.19,E2 22395.19} C_VEL
LIN {X 0,Y 489.688,Z 1150.332,A -85,B 0,C 180,E1 22392.657,E2 22392.657} C_VEL
LIN {X 0,Y 490.761,Z 1142.84,A -85,B 0,C 180,E1 22390.234,E2 22390.234} C_VEL
LIN {X 0,Y 492.154,Z 1134.524,A -85,B 0,C 180,E1 22387.887,E2 22387.887} C_VEL
LIN {X 0,Y 493.846,Z 1125.156,A -85,B 0,C 180,E1 22385.606,E2 22385.606} C_VEL
LIN {X 0,Y 496.097,Z 1113.698,A -85,B 0,C 180,E1 22383.164,E2 22383.164} C_VEL
LIN {X 0,Y 499.065,Z 1098.925,A -85,B 0,C 180,E1 22380.473,E2 22380.473} C_VEL
LIN {X 0,Y 501.781,Z 1085.733,A -85,B 0,C 180,E1 22378.396,E2 22378.396} C_VEL
LIN {X 0,Y 504.667,Z 1071.797,A -85,B 0,C 180,E1 22376.444,E2 22376.444} C_VEL
LIN {X 0,Y 507.746,Z 1056.458,A -85,B 0,C 180,E1 22374.555,E2 22374.555} C_VEL
LIN {X 0,Y 511.811,Z 1035.436,A -85,B 0,C 180,E1 22372.3,E2 22372.3} C_VEL
LIN {X 0,Y 517.602,Z 1005.874,A -85,B 0,C 180,E1 22369.531,E2 22369.531} C_VEL
LIN {X 0,Y 521.702,Z 985.583,A -85,B 0,C 180,E1 22367.832,E2 22367.832} C_VEL
LIN {X 0,Y 526.624,Z 960.398,A -85,B 0,C 180,E1 22365.982,E2 22365.982} C_VEL
LIN {X 0,Y 530.502,Z 939.598,A -85,B 0,C 180,E1 22364.652,E2 22364.652} C_VEL
LIN {X 0,Y 534.838,Z 914.74,A -85,B 0,C 180,E1 22363.269,E2 22363.269} C_VEL
LIN {X 0,Y 538.522,Z 891.13,A -85,B 0,C 180,E1 22362.161,E2 22362.161} C_VEL
LIN {X 0,Y 542.017,Z 866.579,A -85,B 0,C 180,E1 22361.182,E2 22361.182} C_VEL
LIN {X 0,Y 545.115,Z 840.563,A -85,B 0,C 180,E1 22360.351,E2 22360.351} C_VEL
LIN {X 0,Y 547.404,Z 817.702,A -85,B 0,C 180,E1 22359.765,E2 22359.765} C_VEL
LIN {X 0,Y 558.151,Z 694.703,A -85,B 0,C 180,E1 22357.272,E2 22357.272} C_VEL
LIN {X 0,Y 566.683,Z 590.521,A -85,B 0,C 180,E1 22355.353,E2 22355.353} C_VEL
LIN {X 0,Y 572.807,Z 501.469,A -85,B 0,C 180,E1 22353.849,E2 22353.849} C_VEL
LIN {X 0,Y 575.301,Z 456.301,A -85,B 0,C 180,E1 22353.135,E2 22353.135} C_VEL
LIN {X 0,Y 565.448,Z 447.118,A -85,B 0,C 180,E1 22351.325,E2 22351.325} C_VEL
LIN {X 0,Y 557.841,Z 440.394,A -85,B 0,C 180,E1 22349.828,E2 22349.828} C_VEL
LIN {X 0,Y 550.99,Z 434.594,A -85,B 0,C 180,E1 22348.389,E2 22348.389} C_VEL
LIN {X 0,Y 542.355,Z 427.589,A -85,B 0,C 180,E1 22346.379,E2 22346.379} C_VEL
LIN {X 0,Y 540.075,Z 422.967,A -85,B 0,C 180,E1 22343.456,E2 22343.456} C_VEL
LIN {X 0,Y 537.903,Z 418.355,A -85,B 0,C 180,E1 22339.097,E2 22339.097} C_VEL
LIN {X 0,Y 536.726,Z 417.151,A -85,B 0,C 180,E1 22334.566,E2 22334.566} C_VEL
LIN {X 0,Y 537.39,Z 417.887,A -85,B 0,C 180,E1 22330.506,E2 22330.506} C_VEL
LIN {X 0,Y 538.243,Z 418.942,A -85,B 0,C 180,E1 22328.547,E2 22328.547} C_VEL
LIN {X 0,Y 540.757,Z 423.846,A -85,B 0,C 180,E1 22324.242,E2 22324.242} C_VEL
LIN {X 0,Y 543.269,Z 428.926,A -85,B 0,C 180,E1 22321.266,E2 22321.266} C_VEL
LIN {X 0,Y 545.828,Z 434.034,A -85,B 0,C 180,E1 22318.845,E2 22318.845} C_VEL
LIN {X 0,Y 548.238,Z 438.934,A -85,B 0,C 180,E1 22316.863,E2 22316.863} C_VEL
LIN {X 0,Y 550.933,Z 444.416,A -85,B 0,C 180,E1 22314.898,E2 22314.898} C_VEL
LIN {X 0,Y 554.695,Z 452.235,A -85,B 0,C 180,E1 22312.439,E2 22312.439} C_VEL
LIN {X 0,Y 559.554,Z 462.647,A -85,B 0,C 180,E1 22309.602,E2 22309.602} C_VEL
LIN {X 0,Y 564.948,Z 475.156,A -85,B 0,C 180,E1 22306.698,E2 22306.698} C_VEL
LIN {X 0,Y 566.189,Z 478.229,A -85,B 0,C 180,E1 22306.051,E2 22306.051} C_VEL
LIN {X 0,Y 559.295,Z 512.085,A -85,B 0,C 180,E1 22303.022,E2 22303.022} C_VEL
LIN {X 0,Y 552.086,Z 550.012,A -85,B 0,C 180,E1 22299.762,E2 22299.762} C_VEL
LIN {X 0,Y 545.217,Z 588.711,A -85,B 0,C 180,E1 22296.549,E2 22296.549} C_VEL
LIN {X 0,Y 541.346,Z 615.185,A -85,B 0,C 180,E1 22294.332,E2 22294.332} C_VEL
LIN {X 0,Y 540.333,Z 634.898,A -85,B 0,C 180,E1 22292.503,E2 22292.503} C_VEL
LIN {X 0,Y 541.342,Z 652.598,A -85,B 0,C 180,E1 22290.694,E2 22290.694} C_VEL
LIN {X 0,Y 544.31,Z 668.921,A -85,B 0,C 180,E1 22288.87,E2 22288.87} C_VEL
LIN {X 0,Y 549.255,Z 684.181,A -85,B 0,C 180,E1 22287.022,E2 22287.022} C_VEL
LIN {X 0,Y 556.382,Z 698.453,A -85,B 0,C 180,E1 22285.146,E2 22285.146} C_VEL
LIN {X 0,Y 565.037,Z 710.854,A -85,B 0,C 180,E1 22283.39,E2 22283.39} C_VEL
LIN {X 0,Y 570.256,Z 717.045,A -85,B 0,C 180,E1 22282.484,E2 22282.484} C_VEL
LIN {X 0,Y 565.191,Z 745.221,A -85,B 0,C 180,E1 22282.586,E2 22282.586} C_VEL
LIN {X 0,Y 562.28,Z 769.184,A -85,B 0,C 180,E1 22282.495,E2 22282.495} C_VEL
LIN {X 0,Y 560.782,Z 792.708,A -85,B 0,C 180,E1 22282.153,E2 22282.153} C_VEL
LIN {X 0,Y 557.763,Z 828.278,A -85,B 0,C 180,E1 22281.492,E2 22281.492} C_VEL
LIN {X 0,Y 553.943,Z 860.977,A -85,B 0,C 180,E1 22280.739,E2 22280.739} C_VEL
LIN {X 0,Y 549.812,Z 892.628,A -85,B 0,C 180,E1 22279.798,E2 22279.798} C_VEL
LIN {X 0,Y 545.518,Z 922.958,A -85,B 0,C 180,E1 22278.677,E2 22278.677} C_VEL
LIN {X 0,Y 541.171,Z 951.311,A -85,B 0,C 180,E1 22277.413,E2 22277.413} C_VEL
LIN {X 0,Y 536.825,Z 977.42,A -85,B 0,C 180,E1 22276.043,E2 22276.043} C_VEL
LIN {X 0,Y 532.248,Z 1002.902,A -85,B 0,C 180,E1 22274.482,E2 22274.482} C_VEL
LIN {X 0,Y 527.809,Z 1025.973,A -85,B 0,C 180,E1 22272.848,E2 22272.848} C_VEL
LIN {X 0,Y 523.52,Z 1045.971,A -85,B 0,C 180,E1 22271.191,E2 22271.191} C_VEL
LIN {X 0,Y 519.145,Z 1064.129,A -85,B 0,C 180,E1 22269.435,E2 22269.435} C_VEL
LIN {X 0,Y 514.73,Z 1080.549,A -85,B 0,C 180,E1 22267.574,E2 22267.574} C_VEL
LIN {X 0,Y 509.764,Z 1097.069,A -85,B 0,C 180,E1 22265.352,E2 22265.352} C_VEL
LIN {X 0,Y 504.702,Z 1113.816,A -85,B 0,C 180,E1 22262.739,E2 22262.739} C_VEL
LIN {X 0,Y 499.941,Z 1130.664,A -85,B 0,C 180,E1 22259.734,E2 22259.734} C_VEL
LIN {X 0,Y 495.932,Z 1146.543,A -85,B 0,C 180,E1 22256.458,E2 22256.458} C_VEL
LIN {X 0,Y 492.971,Z 1160.484,A -85,B 0,C 180,E1 22253.17,E2 22253.17} C_VEL
LIN {X 0,Y 490.792,Z 1172.872,A -85,B 0,C 180,E1 22249.74,E2 22249.74} C_VEL
LIN {X 0,Y 489.459,Z 1182.256,A -85,B 0,C 180,E1 22246.644,E2 22246.644} C_VEL
LIN {X 0,Y 488.654,Z 1189.808,A -85,B 0,C 180,E1 22243.601,E2 22243.601} C_VEL
LIN {X 0,Y 488.187,Z 1195.946,A -85,B 0,C 180,E1 22240.501,E2 22240.501} C_VEL
LIN {X 0,Y 487.992,Z 1200.348,A -85,B 0,C 180,E1 22237.534,E2 22237.534} C_VEL
LIN {X 0,Y 487.92,Z 1203.226,A -85,B 0,C 180,E1 22234.583,E2 22234.583} C_VEL
LIN {X 0,Y 487.908,Z 1204.757,A -85,B 0,C 180,E1 22231.643,E2 22231.643} C_VEL
LIN {X 0,Y 487.913,Z 1204.828,A -85,B 0,C 180,E1 22228.824,E2 22228.824} C_VEL
LIN {X 0,Y 487.916,Z 1203.577,A -85,B 0,C 180,E1 22225.886,E2 22225.886} C_VEL
LIN {X 0,Y 487.965,Z 1201.024,A -85,B 0,C 180,E1 22223.055,E2 22223.055} C_VEL
LIN {X 0,Y 488.132,Z 1196.92,A -85,B 0,C 180,E1 22220.091,E2 22220.091} C_VEL
LIN {X 0,Y 488.508,Z 1191.404,A -85,B 0,C 180,E1 22217.107,E2 22217.107} C_VEL
LIN {X 0,Y 489.218,Z 1184.246,A -85,B 0,C 180,E1 22214.104,E2 22214.104} C_VEL
LIN {X 0,Y 490.441,Z 1175.104,A -85,B 0,C 180,E1 22210.96,E2 22210.96} C_VEL
LIN {X 0,Y 492.264,Z 1164.146,A -85,B 0,C 180,E1 22207.801,E2 22207.801} C_VEL
LIN {X 0,Y 494.92,Z 1151.157,A -85,B 0,C 180,E1 22204.566,E2 22204.566} C_VEL
LIN {X 0,Y 498.97,Z 1134.38,A -85,B 0,C 180,E1 22200.99,E2 22200.99} C_VEL
LIN {X 0,Y 503.264,Z 1118.687,A -85,B 0,C 180,E1 22198.095,E2 22198.095} C_VEL
LIN {X 0,Y 508.551,Z 1101.07,A -85,B 0,C 180,E1 22195.236,E2 22195.236} C_VEL
LIN {X 0,Y 513.785,Z 1083.691,A -85,B 0,C 180,E1 22192.823,E2 22192.823} C_VEL
LIN {X 0,Y 518.062,Z 1068.352,A -85,B 0,C 180,E1 22191.008,E2 22191.008} C_VEL
LIN {X 0,Y 522.516,Z 1050.216,A -85,B 0,C 180,E1 22189.193,E2 22189.193} C_VEL
LIN {X 0,Y 526.865,Z 1030.376,A -85,B 0,C 180,E1 22187.497,E2 22187.497} C_VEL
LIN {X 0,Y 532.109,Z 1003.671,A -85,B 0,C 180,E1 22185.567,E2 22185.567} C_VEL
LIN {X 0,Y 536.839,Z 977.423,A -85,B 0,C 180,E1 22183.955,E2 22183.955} C_VEL
LIN {X 0,Y 541.368,Z 950.141,A -85,B 0,C 180,E1 22182.528,E2 22182.528} C_VEL
LIN {X 0,Y 545.815,Z 921.07,A -85,B 0,C 180,E1 22181.243,E2 22181.243} C_VEL
LIN {X 0,Y 550.076,Z 890.773,A -85,B 0,C 180,E1 22180.139,E2 22180.139} C_VEL
LIN {X 0,Y 554.15,Z 859.209,A -85,B 0,C 180,E1 22179.217,E2 22179.217} C_VEL
LIN {X 0,Y 558.05,Z 825.32,A -85,B 0,C 180,E1 22178.449,E2 22178.449} C_VEL
LIN {X 0,Y 560.96,Z 789.569,A -85,B 0,C 180,E1 22177.796,E2 22177.796} C_VEL
LIN {X 0,Y 563.892,Z 727.96,A -85,B 0,C 180,E1 22176.9,E2 22176.9} C_VEL
LIN {X 0,Y 565.579,Z 701.586,A -85,B 0,C 180,E1 22176.538,E2 22176.538} C_VEL
LIN {X 0,Y 569.745,Z 662.582,A -85,B 0,C 180,E1 22175.871,E2 22175.871} C_VEL
LIN {X 0,Y 574.723,Z 617.013,A -85,B 0,C 180,E1 22175.107,E2 22175.107} C_VEL
LIN {X 0,Y 576.796,Z 599.78,A -85,B 0,C 180,E1 22174.843,E2 22174.843} C_VEL
LIN {X 0,Y 580.276,Z 567.859,A -85,B 0,C 180,E1 22174.307,E2 22174.307} C_VEL
LIN {X 0,Y 583.639,Z 542.131,A -85,B 0,C 180,E1 22173.95,E2 22173.95} C_VEL
LIN {X 0,Y 586.737,Z 513.218,A -85,B 0,C 180,E1 22173.457,E2 22173.457} C_VEL
LIN {X 0,Y 591.355,Z 479.514,A -85,B 0,C 180,E1 22173.021,E2 22173.021} C_VEL
LIN {X 0,Y 591.206,Z 478.481,A -85,B 0,C 180,E1 22172.968,E2 22172.968} C_VEL
LIN {X 0,Y 579.739,Z 459.483,A -85,B 0,C 180,E1 22170.67,E2 22170.67} C_VEL
LIN {X 0,Y 569.57,Z 443.848,A -85,B 0,C 180,E1 22168.465,E2 22168.465} C_VEL
LIN {X 0,Y 560.778,Z 430.86,A -85,B 0,C 180,E1 22166.387,E2 22166.387} C_VEL
LIN {X 0,Y 550.566,Z 416.496,A -85,B 0,C 180,E1 22163.72,E2 22163.72} C_VEL
LIN {X 0,Y 542.604,Z 405.915,A -85,B 0,C 180,E1 22161.4,E2 22161.4} C_VEL
LIN {X 0,Y 537.707,Z 399.749,A -85,B 0,C 180,E1 22159.838,E2 22159.838} C_VEL
LIN {X 0,Y 533.593,Z 394.401,A -85,B 0,C 180,E1 22158.406,E2 22158.406} C_VEL
LIN {X 0,Y 532.617,Z 393.783,A -85,B 0,C 180,E1 22158.087,E2 22158.087} C_VEL
LIN {X 0,Y 528.818,Z 403.066,A -85,B 0,C 180,E1 22157.51,E2 22157.51} C_VEL
LIN {X 0,Y 527.14,Z 406.824,A -85,B 0,C 180,E1 22157.226,E2 22157.226} C_VEL
LIN {X 0,Y 522.833,Z 419.465,A -85,B 0,C 180,E1 22156.663,E2 22156.663} C_VEL
LIN {X 0,Y 519.434,Z 427.821,A -85,B 0,C 180,E1 22156.093,E2 22156.093} C_VEL
LIN {X 0,Y 518.151,Z 430.716,A -85,B 0,C 180,E1 22155.853,E2 22155.853} C_VEL
LIN {X 0,Y 514.054,Z 443.37,A -85,B 0,C 180,E1 22155.3,E2 22155.3} C_VEL
LIN {X 0,Y 510.948,Z 451.445,A -85,B 0,C 180,E1 22154.753,E2 22154.753} C_VEL
LIN {X 0,Y 509.389,Z 454.958,A -85,B 0,C 180,E1 22154.428,E2 22154.428} C_VEL
LIN {X 0,Y 505.429,Z 467.697,A -85,B 0,C 180,E1 22153.866,E2 22153.866} C_VEL
LIN {X 0,Y 502.648,Z 475.252,A -85,B 0,C 180,E1 22153.341,E2 22153.341} C_VEL
LIN {X 0,Y 501.274,Z 478.224,A -85,B 0,C 180,E1 22152.983,E2 22152.983} C_VEL
LIN {X 0,Y 500.742,Z 552.82,A -85,B 0,C 180,E1 22149.975,E2 22149.975} C_VEL
LIN {X 0,Y 499.884,Z 621.852,A -85,B 0,C 180,E1 22147.124,E2 22147.124} C_VEL
LIN {X 0,Y 498.649,Z 699.222,A -85,B 0,C 180,E1 22143.881,E2 22143.881} C_VEL
LIN {X 0,Y 497.161,Z 776.951,A -85,B 0,C 180,E1 22140.547,E2 22140.547} C_VEL
LIN {X 0,Y 495.601,Z 851.822,A -85,B 0,C 180,E1 22137.277,E2 22137.277} C_VEL
LIN {X 0,Y 494.145,Z 870.375,A -85,B 0,C 180,E1 22136.529,E2 22136.529} C_VEL
LIN {X 0,Y 492.877,Z 975.332,A -85,B 0,C 180,E1 22134.81,E2 22134.81} C_VEL
LIN {X 0,Y 493.014,Z 992.285,A -85,B 0,C 180,E1 22134.432,E2 22134.432} C_VEL
LIN {X 0,Y 492.963,Z 1005.294,A -85,B 0,C 180,E1 22133.946,E2 22133.946} C_VEL
LIN {X 0,Y 492.8,Z 1016.912,A -85,B 0,C 180,E1 22133.359,E2 22133.359} C_VEL
LIN {X 0,Y 492.54,Z 1028.649,A -85,B 0,C 180,E1 22132.593,E2 22132.593} C_VEL
LIN {X 0,Y 492.134,Z 1041.119,A -85,B 0,C 180,E1 22131.529,E2 22131.529} C_VEL
LIN {X 0,Y 491.735,Z 1050.402,A -85,B 0,C 180,E1 22130.52,E2 22130.52} C_VEL
LIN {X 0,Y 491.389,Z 1057.613,A -85,B 0,C 180,E1 22129.566,E2 22129.566} C_VEL
LIN {X 0,Y 491.036,Z 1064.303,A -85,B 0,C 180,E1 22128.489,E2 22128.489} C_VEL
LIN {X 0,Y 490.693,Z 1070.297,A -85,B 0,C 180,E1 22127.287,E2 22127.287} C_VEL
LIN {X 0,Y 490.371,Z 1075.85,A -85,B 0,C 180,E1 22125.837,E2 22125.837} C_VEL
LIN {X 0,Y 490.099,Z 1079.874,A -85,B 0,C 180,E1 22124.256,E2 22124.256} C_VEL
LIN {X 0,Y 489.948,Z 1081.936,A -85,B 0,C 180,E1 22122.91,E2 22122.91} C_VEL
LIN {X 0,Y 489.859,Z 1082.811,A -85,B 0,C 180,E1 22121.556,E2 22121.556} C_VEL
LIN {X 0,Y 489.83,Z 1082.496,A -85,B 0,C 180,E1 22120.193,E2 22120.193} C_VEL
LIN {X 0,Y 489.865,Z 1080.8,A -85,B 0,C 180,E1 22118.695,E2 22118.695} C_VEL
LIN {X 0,Y 490.026,Z 1076.867,A -85,B 0,C 180,E1 22116.935,E2 22116.935} C_VEL
LIN {X 0,Y 490.224,Z 1072.146,A -85,B 0,C 180,E1 22115.54,E2 22115.54} C_VEL
LIN {X 0,Y 490.494,Z 1066.482,A -85,B 0,C 180,E1 22114.265,E2 22114.265} C_VEL
LIN {X 0,Y 490.894,Z 1058.525,A -85,B 0,C 180,E1 22112.854,E2 22112.854} C_VEL
LIN {X 0,Y 491.339,Z 1048.881,A -85,B 0,C 180,E1 22111.539,E2 22111.539} C_VEL
LIN {X 0,Y 491.753,Z 1039.301,A -85,B 0,C 180,E1 22110.49,E2 22110.49} C_VEL
LIN {X 0,Y 492.149,Z 1028.668,A -85,B 0,C 180,E1 22109.542,E2 22109.542} C_VEL
LIN {X 0,Y 492.578,Z 1014.427,A -85,B 0,C 180,E1 22108.554,E2 22108.554} C_VEL
LIN {X 0,Y 492.82,Z 1002.263,A -85,B 0,C 180,E1 22107.922,E2 22107.922} C_VEL
LIN {X 0,Y 492.945,Z 989.931,A -85,B 0,C 180,E1 22107.442,E2 22107.442} C_VEL
LIN {X 0,Y 492.967,Z 974.867,A -85,B 0,C 180,E1 22107.049,E2 22107.049} C_VEL
LIN {X 0,Y 494.249,Z 864.666,A -85,B 0,C 180,E1 22105.285,E2 22105.285} C_VEL
LIN {X 0,Y 494.882,Z 865.792,A -85,B 0,C 180,E1 22105.117,E2 22105.117} C_VEL
LIN {X 0,Y 496.007,Z 865.853,A -85,B 0,C 180,E1 22104.933,E2 22104.933} C_VEL
LIN {X 0,Y 498.097,Z 863.896,A -85,B 0,C 180,E1 22104.715,E2 22104.715} C_VEL
LIN {X 0,Y 503.348,Z 856.422,A -85,B 0,C 180,E1 22104.316,E2 22104.316} C_VEL
LIN {X 0,Y 503.686,Z 855.904,A -85,B 0,C 180,E1 22104.293,E2 22104.293} C_VEL
LIN {X 0,Y 507.075,Z 854.22,A -85,B 0,C 180,E1 22103.872,E2 22103.872} C_VEL
LIN {X 0,Y 511.09,Z 850.284,A -85,B 0,C 180,E1 22103.488,E2 22103.488} C_VEL
LIN {X 0,Y 514,Z 846.497,A -85,B 0,C 180,E1 22103.26,E2 22103.26} C_VEL
LIN {X 0,Y 518.404,Z 843.36,A -85,B 0,C 180,E1 22102.794,E2 22102.794} C_VEL
LIN {X 0,Y 523.237,Z 837.915,A -85,B 0,C 180,E1 22102.387,E2 22102.387} C_VEL
LIN {X 0,Y 524.735,Z 836.139,A -85,B 0,C 180,E1 22102.26,E2 22102.26} C_VEL
LIN {X 0,Y 529.862,Z 831.921,A -85,B 0,C 180,E1 22101.759,E2 22101.759} C_VEL
LIN {X 0,Y 535.596,Z 825.278,A -85,B 0,C 180,E1 22101.288,E2 22101.288} C_VEL
LIN {X 0,Y 541.413,Z 820.169,A -85,B 0,C 180,E1 22100.762,E2 22100.762} C_VEL
LIN {X 0,Y 546.358,Z 814.567,A -85,B 0,C 180,E1 22100.373,E2 22100.373} C_VEL
LIN {X 0,Y 547.802,Z 813.651,A -85,B 0,C 180,E1 22100.235,E2 22100.235} C_VEL
LIN {X 0,Y 545.311,Z 838.728,A -85,B 0,C 180,E1 22099.61,E2 22099.61} C_VEL
LIN {X 0,Y 542.31,Z 864.151,A -85,B 0,C 180,E1 22098.814,E2 22098.814} C_VEL
LIN {X 0,Y 538.657,Z 890.234,A -85,B 0,C 180,E1 22097.788,E2 22097.788} C_VEL
LIN {X 0,Y 535.103,Z 912.941,A -85,B 0,C 180,E1 22096.73,E2 22096.73} C_VEL
LIN {X 0,Y 530.554,Z 939.289,A -85,B 0,C 180,E1 22095.277,E2 22095.277} C_VEL
LIN {X 0,Y 528.877,Z 948.63,A -85,B 0,C 180,E1 22094.707,E2 22094.707} C_VEL
LIN {X 0,Y 526.868,Z 955.386,A -85,B 0,C 180,E1 22094.352,E2 22094.352} C_VEL
LIN {X 0,Y 518.772,Z 972.483,A -85,B 0,C 180,E1 22093.592,E2 22093.592} C_VEL
LIN {X 0,Y 516.685,Z 978.933,A -85,B 0,C 180,E1 22093.18,E2 22093.18} C_VEL
LIN {X 0,Y 511.614,Z 1002.841,A -85,B 0,C 180,E1 22091.196,E2 22091.196} C_VEL
LIN {X 0,Y 507.431,Z 1022.122,A -85,B 0,C 180,E1 22089.384,E2 22089.384} C_VEL
LIN {X 0,Y 501.99,Z 1047.528,A -85,B 0,C 180,E1 22086.696,E2 22086.696} C_VEL
LIN {X 0,Y 498.298,Z 1066.096,A -85,B 0,C 180,E1 22084.533,E2 22084.533} C_VEL
LIN {X 0,Y 494.79,Z 1083.03,A -85,B 0,C 180,E1 22082.243,E2 22082.243} C_VEL
LIN {X 0,Y 492.254,Z 1095.122,A -85,B 0,C 180,E1 22080.384,E2 22080.384} C_VEL
LIN {X 0,Y 489.821,Z 1106.721,A -85,B 0,C 180,E1 22078.379,E2 22078.379} C_VEL
LIN {X 0,Y 487.627,Z 1117.485,A -85,B 0,C 180,E1 22076.291,E2 22076.291} C_VEL
LIN {X 0,Y 485.766,Z 1127.05,A -85,B 0,C 180,E1 22074.182,E2 22074.182} C_VEL
LIN {X 0,Y 483.749,Z 1138.301,A -85,B 0,C 180,E1 22071.334,E2 22071.334} C_VEL
LIN {X 0,Y 482.173,Z 1147.947,A -85,B 0,C 180,E1 22068.374,E2 22068.374} C_VEL
LIN {X 0,Y 481.189,Z 1155.315,A -85,B 0,C 180,E1 22065.674,E2 22065.674} C_VEL
LIN {X 0,Y 480.566,Z 1161.205,A -85,B 0,C 180,E1 22063.109,E2 22063.109} C_VEL
LIN {X 0,Y 480.204,Z 1166.004,A -85,B 0,C 180,E1 22060.56,E2 22060.56} C_VEL
LIN {X 0,Y 480.02,Z 1169.749,A -85,B 0,C 180,E1 22058.024,E2 22058.024} C_VEL
LIN {X 0,Y 479.933,Z 1172.467,A -85,B 0,C 180,E1 22055.501,E2 22055.501} C_VEL
LIN {X 0,Y 479.912,Z 1174.175,A -85,B 0,C 180,E1 22052.987,E2 22052.987} C_VEL
LIN {X 0,Y 479.895,Z 1174.886,A -85,B 0,C 180,E1 22050.479,E2 22050.479} C_VEL
LIN {X 0,Y 479.911,Z 1174.553,A -85,B 0,C 180,E1 22047.852,E2 22047.852} C_VEL
LIN {X 0,Y 479.92,Z 1173.127,A -85,B 0,C 180,E1 22045.221,E2 22045.221} C_VEL
LIN {X 0,Y 479.982,Z 1170.743,A -85,B 0,C 180,E1 22042.701,E2 22042.701} C_VEL
LIN {X 0,Y 480.133,Z 1167.187,A -85,B 0,C 180,E1 22040.078,E2 22040.078} C_VEL
LIN {X 0,Y 480.438,Z 1162.633,A -85,B 0,C 180,E1 22037.501,E2 22037.501} C_VEL
LIN {X 0,Y 480.978,Z 1157.042,A -85,B 0,C 180,E1 22034.94,E2 22034.94} C_VEL
LIN {X 0,Y 481.818,Z 1150.328,A -85,B 0,C 180,E1 22032.365,E2 22032.365} C_VEL
LIN {X 0,Y 482.893,Z 1143.188,A -85,B 0,C 180,E1 22030.024,E2 22030.024} C_VEL
LIN {X 0,Y 484.332,Z 1134.786,A -85,B 0,C 180,E1 22027.652,E2 22027.652} C_VEL
LIN {X 0,Y 486.097,Z 1125.309,A -85,B 0,C 180,E1 22025.321,E2 22025.321} C_VEL
LIN {X 0,Y 488.298,Z 1114.305,A -85,B 0,C 180,E1 22022.964,E2 22022.964} C_VEL
LIN {X 0,Y 491.495,Z 1098.656,A -85,B 0,C 180,E1 22020.106,E2 22020.106} C_VEL
LIN {X 0,Y 494.13,Z 1086.141,A -85,B 0,C 180,E1 22018.122,E2 22018.122} C_VEL
LIN {X 0,Y 497.076,Z 1071.938,A -85,B 0,C 180,E1 22016.14,E2 22016.14} C_VEL
LIN {X 0,Y 500.774,Z 1053.897,A -85,B 0,C 180,E1 22013.915,E2 22013.915} C_VEL
LIN {X 0,Y 506.87,Z 1024.789,A -85,B 0,C 180,E1 22010.787,E2 22010.787} C_VEL
LIN {X 0,Y 511.315,Z 1004.235,A -85,B 0,C 180,E1 22008.841,E2 22008.841} C_VEL
LIN {X 0,Y 516.009,Z 982.427,A -85,B 0,C 180,E1 22006.996,E2 22006.996} C_VEL
LIN {X 0,Y 520.613,Z 959.747,A -85,B 0,C 180,E1 22005.34,E2 22005.34} C_VEL
LIN {X 0,Y 525.036,Z 937.108,A -85,B 0,C 180,E1 22003.885,E2 22003.885} C_VEL
LIN {X 0,Y 529.54,Z 911.68,A -85,B 0,C 180,E1 22002.497,E2 22002.497} C_VEL
LIN {X 0,Y 533.315,Z 888.481,A -85,B 0,C 180,E1 22001.418,E2 22001.418} C_VEL
LIN {X 0,Y 537.139,Z 861.336,A -85,B 0,C 180,E1 22000.374,E2 22000.374} C_VEL
LIN {X 0,Y 539.913,Z 838.701,A -85,B 0,C 180,E1 21999.67,E2 21999.67} C_VEL
LIN {X 0,Y 542.724,Z 810.754,A -85,B 0,C 180,E1 21998.979,E2 21998.979} C_VEL
LIN {X 0,Y 554.322,Z 683.234,A -85,B 0,C 180,E1 21996.391,E2 21996.391} C_VEL
LIN {X 0,Y 562.441,Z 586.726,A -85,B 0,C 180,E1 21994.612,E2 21994.612} C_VEL
LIN {X 0,Y 568.441,Z 501.549,A -85,B 0,C 180,E1 21993.173,E2 21993.173} C_VEL
LIN {X 0,Y 570.714,Z 461.53,A -85,B 0,C 180,E1 21992.538,E2 21992.538} C_VEL
LIN {X 0,Y 562.411,Z 453.879,A -85,B 0,C 180,E1 21990.977,E2 21990.977} C_VEL
LIN {X 0,Y 555.344,Z 447.599,A -85,B 0,C 180,E1 21989.56,E2 21989.56} C_VEL
LIN {X 0,Y 548.772,Z 441.988,A -85,B 0,C 180,E1 21988.159,E2 21988.159} C_VEL
LIN {X 0,Y 540.036,Z 435.044,A -85,B 0,C 180,E1 21986.146,E2 21986.146} C_VEL
LIN {X 0,Y 537.075,Z 432.851,A -85,B 0,C 180,E1 21985.353,E2 21985.353} C_VEL
LIN {X 0,Y 535.809,Z 429.727,A -85,B 0,C 180,E1 21983.421,E2 21983.421} C_VEL
LIN {X 0,Y 533.663,Z 425.136,A -85,B 0,C 180,E1 21979.027,E2 21979.027} C_VEL
LIN {X 0,Y 532.538,Z 423.967,A -85,B 0,C 180,E1 21974.572,E2 21974.572} C_VEL
LIN {X 0,Y 533.208,Z 424.711,A -85,B 0,C 180,E1 21970.48,E2 21970.48} C_VEL
LIN {X 0,Y 534.014,Z 425.704,A -85,B 0,C 180,E1 21968.615,E2 21968.615} C_VEL
LIN {X 0,Y 536.47,Z 430.644,A -85,B 0,C 180,E1 21964.276,E2 21964.276} C_VEL
LIN {X 0,Y 538.952,Z 435.76,A -85,B 0,C 180,E1 21961.276,E2 21961.276} C_VEL
LIN {X 0,Y 541.387,Z 440.634,A -85,B 0,C 180,E1 21958.942,E2 21958.942} C_VEL
LIN {X 0,Y 543.765,Z 445.545,A -85,B 0,C 180,E1 21956.943,E2 21956.943} C_VEL
LIN {X 0,Y 547.242,Z 452.479,A -85,B 0,C 180,E1 21954.443,E2 21954.443} C_VEL
LIN {X 0,Y 551.488,Z 461.715,A -85,B 0,C 180,E1 21951.66,E2 21951.66} C_VEL
LIN {X 0,Y 556.371,Z 472.699,A -85,B 0,C 180,E1 21948.808,E2 21948.808} C_VEL
LIN {X 0,Y 560.786,Z 483.111,A -85,B 0,C 180,E1 21946.44,E2 21946.44} C_VEL
LIN {X 0,Y 553.576,Z 517.314,A -85,B 0,C 180,E1 21943.364,E2 21943.364} C_VEL
LIN {X 0,Y 545.845,Z 556.63,A -85,B 0,C 180,E1 21939.968,E2 21939.968} C_VEL
LIN {X 0,Y 538.809,Z 594.956,A -85,B 0,C 180,E1 21936.769,E2 21936.769} C_VEL
LIN {X 0,Y 535.206,Z 619.601,A -85,B 0,C 180,E1 21934.67,E2 21934.67} C_VEL
LIN {X 0,Y 534.179,Z 639.174,A -85,B 0,C 180,E1 21932.824,E2 21932.824} C_VEL
LIN {X 0,Y 535.166,Z 657.04,A -85,B 0,C 180,E1 21930.97,E2 21930.97} C_VEL
LIN {X 0,Y 538.041,Z 673.179,A -85,B 0,C 180,E1 21929.142,E2 21929.142} C_VEL
LIN {X 0,Y 543.025,Z 688.818,A -85,B 0,C 180,E1 21927.224,E2 21927.224} C_VEL
LIN {X 0,Y 546.235,Z 695.765,A -85,B 0,C 180,E1 21926.361,E2 21926.361} C_VEL
LIN {X 0,Y 554.513,Z 708.788,A -85,B 0,C 180,E1 21924.822,E2 21924.822} C_VEL
LIN {X 0,Y 564.35,Z 720.741,A -85,B 0,C 180,E1 21923.192,E2 21923.192} C_VEL
LIN {X 0,Y 564.415,Z 721.568,A -85,B 0,C 180,E1 21923.167,E2 21923.167} C_VEL
LIN {X 0,Y 559.57,Z 750.591,A -85,B 0,C 180,E1 21923.234,E2 21923.234} C_VEL
LIN {X 0,Y 557.132,Z 772.331,A -85,B 0,C 180,E1 21923.113,E2 21923.113} C_VEL
LIN {X 0,Y 554.55,Z 808.301,A -85,B 0,C 180,E1 21922.517,E2 21922.517} C_VEL
LIN {X 0,Y 550.677,Z 844.203,A -85,B 0,C 180,E1 21921.775,E2 21921.775} C_VEL
LIN {X 0,Y 546.477,Z 876.724,A -85,B 0,C 180,E1 21920.915,E2 21920.915} C_VEL
LIN {X 0,Y 542.154,Z 907.219,A -85,B 0,C 180,E1 21919.897,E2 21919.897} C_VEL
LIN {X 0,Y 537.668,Z 936.555,A -85,B 0,C 180,E1 21918.701,E2 21918.701} C_VEL
LIN {X 0,Y 533.011,Z 964.668,A -85,B 0,C 180,E1 21917.335,E2 21917.335} C_VEL
LIN {X 0,Y 528.3,Z 991.027,A -85,B 0,C 180,E1 21915.83,E2 21915.83} C_VEL
LIN {X 0,Y 523.437,Z 1016.289,A -85,B 0,C 180,E1 21914.147,E2 21914.147} C_VEL
LIN {X 0,Y 519.115,Z 1037.205,A -85,B 0,C 180,E1 21912.535,E2 21912.535} C_VEL
LIN {X 0,Y 514.553,Z 1056.955,A -85,B 0,C 180,E1 21910.76,E2 21910.76} C_VEL
LIN {X 0,Y 509.93,Z 1075.018,A -85,B 0,C 180,E1 21908.861,E2 21908.861} C_VEL
LIN {X 0,Y 505.309,Z 1091.493,A -85,B 0,C 180,E1 21906.836,E2 21906.836} C_VEL
LIN {X 0,Y 500.968,Z 1105.51,A -85,B 0,C 180,E1 21904.806,E2 21904.806} C_VEL
LIN {X 0,Y 495.916,Z 1121.362,A -85,B 0,C 180,E1 21902.132,E2 21902.132} C_VEL
LIN {X 0,Y 490.781,Z 1138.674,A -85,B 0,C 180,E1 21898.736,E2 21898.736} C_VEL
LIN {X 0,Y 487.11,Z 1152.838,A -85,B 0,C 180,E1 21895.533,E2 21895.533} C_VEL
LIN {X 0,Y 484.233,Z 1166.199,A -85,B 0,C 180,E1 21892.072,E2 21892.072} C_VEL
LIN {X 0,Y 482.329,Z 1177.055,A -85,B 0,C 180,E1 21888.741,E2 21888.741} C_VEL
LIN {X 0,Y 481.175,Z 1185.485,A -85,B 0,C 180,E1 21885.671,E2 21885.671} C_VEL
LIN {X 0,Y 480.444,Z 1192.604,A -85,B 0,C 180,E1 21882.498,E2 21882.498} C_VEL
LIN {X 0,Y 480.1,Z 1197.903,A -85,B 0,C 180,E1 21879.468,E2 21879.468} C_VEL
LIN {X 0,Y 479.958,Z 1201.644,A -85,B 0,C 180,E1 21876.458,E2 21876.458} C_VEL
LIN {X 0,Y 479.916,Z 1204.027,A -85,B 0,C 180,E1 21873.462,E2 21873.462} C_VEL
LIN {X 0,Y 479.898,Z 1204.899,A -85,B 0,C 180,E1 21870.715,E2 21870.715} C_VEL
LIN {X 0,Y 479.909,Z 1204.554,A -85,B 0,C 180,E1 21867.73,E2 21867.73} C_VEL
LIN {X 0,Y 479.931,Z 1202.87,A -85,B 0,C 180,E1 21864.859,E2 21864.859} C_VEL
LIN {X 0,Y 480.026,Z 1199.544,A -85,B 0,C 180,E1 21861.735,E2 21861.735} C_VEL
LIN {X 0,Y 480.271,Z 1194.888,A -85,B 0,C 180,E1 21858.694,E2 21858.694} C_VEL
LIN {X 0,Y 480.822,Z 1188.703,A -85,B 0,C 180,E1 21855.671,E2 21855.671} C_VEL
LIN {X 0,Y 481.793,Z 1180.589,A -85,B 0,C 180,E1 21852.486,E2 21852.486} C_VEL
LIN {X 0,Y 483.439,Z 1170.398,A -85,B 0,C 180,E1 21849.16,E2 21849.16} C_VEL
LIN {X 0,Y 485.643,Z 1159.231,A -85,B 0,C 180,E1 21846.07,E2 21846.07} C_VEL
LIN {X 0,Y 489.243,Z 1144.414,A -85,B 0,C 180,E1 21842.498,E2 21842.498} C_VEL
LIN {X 0,Y 493.965,Z 1127.738,A -85,B 0,C 180,E1 21839.058,E2 21839.058} C_VEL
LIN {X 0,Y 499.055,Z 1111.484,A -85,B 0,C 180,E1 21836.151,E2 21836.151} C_VEL
LIN {X 0,Y 503.754,Z 1096.709,A -85,B 0,C 180,E1 21833.877,E2 21833.877} C_VEL
LIN {X 0,Y 508.264,Z 1081.079,A -85,B 0,C 180,E1 21831.849,E2 21831.849} C_VEL
LIN {X 0,Y 513.094,Z 1062.817,A -85,B 0,C 180,E1 21829.831,E2 21829.831} C_VEL
LIN {X 0,Y 517.622,Z 1044.023,A -85,B 0,C 180,E1 21828.048,E2 21828.048} C_VEL
LIN {X 0,Y 522.029,Z 1023.62,A -85,B 0,C 180,E1 21826.388,E2 21826.388} C_VEL
LIN {X 0,Y 527.078,Z 997.486,A -85,B 0,C 180,E1 21824.58,E2 21824.58} C_VEL
LIN {X 0,Y 531.793,Z 971.701,A -85,B 0,C 180,E1 21823.041,E2 21823.041} C_VEL
LIN {X 0,Y 536.682,Z 942.738,A -85,B 0,C 180,E1 21821.579,E2 21821.579} C_VEL
LIN {X 0,Y 541.202,Z 913.672,A -85,B 0,C 180,E1 21820.349,E2 21820.349} C_VEL
LIN {X 0,Y 545.687,Z 882.405,A -85,B 0,C 180,E1 21819.259,E2 21819.259} C_VEL
LIN {X 0,Y 549.909,Z 850.34,A -85,B 0,C 180,E1 21818.369,E2 21818.369} C_VEL
LIN {X 0,Y 553.837,Z 815.646,A -85,B 0,C 180,E1 21817.626,E2 21817.626} C_VEL
LIN {X 0,Y 556.768,Z 776.785,A -85,B 0,C 180,E1 21816.94,E2 21816.94} C_VEL
LIN {X 0,Y 560.413,Z 705.131,A -85,B 0,C 180,E1 21815.951,E2 21815.951} C_VEL
LIN {X 0,Y 564.305,Z 667.048,A -85,B 0,C 180,E1 21815.299,E2 21815.299} C_VEL
LIN {X 0,Y 566.345,Z 648.299,A -85,B 0,C 180,E1 21814.978,E2 21814.978} C_VEL
LIN {X 0,Y 570.709,Z 610.941,A -85,B 0,C 180,E1 21814.379,E2 21814.379} C_VEL
LIN {X 0,Y 572.113,Z 598.523,A -85,B 0,C 180,E1 21814.174,E2 21814.174} C_VEL
LIN {X 0,Y 575.872,Z 565.456,A -85,B 0,C 180,E1 21813.631,E2 21813.631} C_VEL
LIN {X 0,Y 578.904,Z 542.524,A -85,B 0,C 180,E1 21813.314,E2 21813.314} C_VEL
LIN {X 0,Y 582.125,Z 513.157,A -85,B 0,C 180,E1 21812.815,E2 21812.815} C_VEL
LIN {X 0,Y 586.368,Z 482.879,A -85,B 0,C 180,E1 21812.432,E2 21812.432} C_VEL
LIN {X 0,Y 575.729,Z 465.102,A -85,B 0,C 180,E1 21810.242,E2 21810.242} C_VEL
LIN {X 0,Y 565.517,Z 449.242,A -85,B 0,C 180,E1 21807.969,E2 21807.969} C_VEL
LIN {X 0,Y 556.966,Z 436.59,A -85,B 0,C 180,E1 21805.893,E2 21805.893} C_VEL
LIN {X 0,Y 547.647,Z 423.344,A -85,B 0,C 180,E1 21803.398,E2 21803.398} C_VEL
LIN {X 0,Y 539.965,Z 413.018,A -85,B 0,C 180,E1 21801.111,E2 21801.111} C_VEL
LIN {X 0,Y 535.14,Z 406.865,A -85,B 0,C 180,E1 21799.54,E2 21799.54} C_VEL
LIN {X 0,Y 532.205,Z 403.119,A -85,B 0,C 180,E1 21798.513,E2 21798.513} C_VEL
LIN {X 0,Y 528.634,Z 411.272,A -85,B 0,C 180,E1 21797.95,E2 21797.95} C_VEL
LIN {X 0,Y 524.115,Z 424.154,A -85,B 0,C 180,E1 21797.364,E2 21797.364} C_VEL
LIN {X 0,Y 520.458,Z 432.916,A -85,B 0,C 180,E1 21796.763,E2 21796.763} C_VEL
LIN {X 0,Y 519.415,Z 435.417,A -85,B 0,C 180,E1 21796.587,E2 21796.587} C_VEL
LIN {X 0,Y 515.155,Z 448.152,A -85,B 0,C 180,E1 21796.013,E2 21796.013} C_VEL
LIN {X 0,Y 511.765,Z 456.682,A -85,B 0,C 180,E1 21795.424,E2 21795.424} C_VEL
LIN {X 0,Y 510.49,Z 459.673,A -85,B 0,C 180,E1 21795.18,E2 21795.18} C_VEL
LIN {X 0,Y 506.364,Z 472.503,A -85,B 0,C 180,E1 21794.593,E2 21794.593} C_VEL
LIN {X 0,Y 503.38,Z 480.348,A -85,B 0,C 180,E1 21794.039,E2 21794.039} C_VEL
LIN {X 0,Y 501.985,Z 483.536,A -85,B 0,C 180,E1 21793.734,E2 21793.734} C_VEL
LIN {X 0,Y 497.985,Z 496.546,A -85,B 0,C 180,E1 21793.137,E2 21793.137} C_VEL
LIN {X 0,Y 495.165,Z 504.374,A -85,B 0,C 180,E1 21792.582,E2 21792.582} C_VEL
LIN {X 0,Y 493.911,Z 507.393,A -85,B 0,C 180,E1 21792.236,E2 21792.236} C_VEL
LIN {X 0,Y 493.144,Z 580.983,A -85,B 0,C 180,E1 21789.217,E2 21789.217} C_VEL
LIN {X 0,Y 491.928,Z 659.499,A -85,B 0,C 180,E1 21785.921,E2 21785.921} C_VEL
LIN {X 0,Y 490.392,Z 740.018,A -85,B 0,C 180,E1 21782.483,E2 21782.483} C_VEL
LIN {X 0,Y 488.744,Z 819.027,A -85,B 0,C 180,E1 21779.033,E2 21779.033} C_VEL
LIN {X 0,Y 487.751,Z 855.587,A -85,B 0,C 180,E1 21777.432,E2 21777.432} C_VEL
LIN {X 0,Y 486.461,Z 871.744,A -85,B 0,C 180,E1 21776.776,E2 21776.776} C_VEL
LIN {X 0,Y 485.116,Z 974.949,A -85,B 0,C 180,E1 21775.047,E2 21775.047} C_VEL
LIN {X 0,Y 485.263,Z 992.255,A -85,B 0,C 180,E1 21774.672,E2 21774.672} C_VEL
LIN {X 0,Y 485.203,Z 1006.338,A -85,B 0,C 180,E1 21774.145,E2 21774.145} C_VEL
LIN {X 0,Y 485.028,Z 1018.061,A -85,B 0,C 180,E1 21773.544,E2 21773.544} C_VEL
LIN {X 0,Y 484.765,Z 1029.196,A -85,B 0,C 180,E1 21772.809,E2 21772.809} C_VEL
LIN {X 0,Y 484.33,Z 1042.238,A -85,B 0,C 180,E1 21771.691,E2 21771.691} C_VEL
LIN {X 0,Y 483.914,Z 1051.549,A -85,B 0,C 180,E1 21770.665,E2 21770.665} C_VEL
LIN {X 0,Y 483.528,Z 1059.183,A -85,B 0,C 180,E1 21769.636,E2 21769.636} C_VEL
LIN {X 0,Y 483.161,Z 1065.813,A -85,B 0,C 180,E1 21768.541,E2 21768.541} C_VEL
LIN {X 0,Y 482.796,Z 1071.908,A -85,B 0,C 180,E1 21767.283,E2 21767.283} C_VEL
LIN {X 0,Y 482.413,Z 1077.909,A -85,B 0,C 180,E1 21765.598,E2 21765.598} C_VEL
LIN {X 0,Y 482.165,Z 1081.364,A -85,B 0,C 180,E1 21764.113,E2 21764.113} C_VEL
LIN {X 0,Y 482.018,Z 1083.261,A -85,B 0,C 180,E1 21762.744,E2 21762.744} C_VEL
LIN {X 0,Y 481.931,Z 1083.964,A -85,B 0,C 180,E1 21761.366,E2 21761.366} C_VEL
LIN {X 0,Y 481.921,Z 1083.306,A -85,B 0,C 180,E1 21759.727,E2 21759.727} C_VEL
LIN {X 0,Y 481.987,Z 1080.681,A -85,B 0,C 180,E1 21758.021,E2 21758.021} C_VEL
LIN {X 0,Y 482.131,Z 1077.271,A -85,B 0,C 180,E1 21756.664,E2 21756.664} C_VEL
LIN {X 0,Y 482.334,Z 1072.832,A -85,B 0,C 180,E1 21755.375,E2 21755.375} C_VEL
LIN {X 0,Y 482.633,Z 1066.898,A -85,B 0,C 180,E1 21754.046,E2 21754.046} C_VEL
LIN {X 0,Y 483.091,Z 1058.03,A -85,B 0,C 180,E1 21752.512,E2 21752.512} C_VEL
LIN {X 0,Y 483.508,Z 1049.215,A -85,B 0,C 180,E1 21751.329,E2 21751.329} C_VEL
LIN {X 0,Y 483.941,Z 1039.563,A -85,B 0,C 180,E1 21750.272,E2 21750.272} C_VEL
LIN {X 0,Y 484.406,Z 1027.556,A -85,B 0,C 180,E1 21749.209,E2 21749.209} C_VEL
LIN {X 0,Y 484.782,Z 1014.617,A -85,B 0,C 180,E1 21748.337,E2 21748.337} C_VEL
LIN {X 0,Y 485.023,Z 1002.948,A -85,B 0,C 180,E1 21747.728,E2 21747.728} C_VEL
LIN {X 0,Y 485.156,Z 990.204,A -85,B 0,C 180,E1 21747.23,E2 21747.23} C_VEL
LIN {X 0,Y 485.164,Z 973.711,A -85,B 0,C 180,E1 21746.816,E2 21746.816} C_VEL
LIN {X 0,Y 486.216,Z 883.662,A -85,B 0,C 180,E1 21745.346,E2 21745.346} C_VEL
LIN {X 0,Y 486.817,Z 884.605,A -85,B 0,C 180,E1 21745.18,E2 21745.18} C_VEL
LIN {X 0,Y 487.966,Z 884.639,A -85,B 0,C 180,E1 21744.988,E2 21744.988} C_VEL
LIN {X 0,Y 489.853,Z 883.087,A -85,B 0,C 180,E1 21744.785,E2 21744.785} C_VEL
LIN {X 0,Y 492.834,Z 878.728,A -85,B 0,C 180,E1 21744.596,E2 21744.596} C_VEL
LIN {X 0,Y 495.859,Z 872.903,A -85,B 0,C 180,E1 21744.497,E2 21744.497} C_VEL
LIN {X 0,Y 498.829,Z 870.625,A -85,B 0,C 180,E1 21744.175,E2 21744.175} C_VEL
LIN {X 0,Y 505.477,Z 862.457,A -85,B 0,C 180,E1 21743.669,E2 21743.669} C_VEL
LIN {X 0,Y 509.875,Z 859.364,A -85,B 0,C 180,E1 21743.194,E2 21743.194} C_VEL
LIN {X 0,Y 514.658,Z 854.119,A -85,B 0,C 180,E1 21742.783,E2 21742.783} C_VEL
LIN {X 0,Y 516.043,Z 852.641,A -85,B 0,C 180,E1 21742.665,E2 21742.665} C_VEL
LIN {X 0,Y 521.206,Z 848.47,A -85,B 0,C 180,E1 21742.163,E2 21742.163} C_VEL
LIN {X 0,Y 526.847,Z 842.238,A -85,B 0,C 180,E1 21741.709,E2 21741.709} C_VEL
LIN {X 0,Y 532.741,Z 837.214,A -85,B 0,C 180,E1 21741.18,E2 21741.18} C_VEL
LIN {X 0,Y 537.977,Z 831.373,A -85,B 0,C 180,E1 21740.773,E2 21740.773} C_VEL
LIN {X 0,Y 540.954,Z 829,A -85,B 0,C 180,E1 21740.504,E2 21740.504} C_VEL
LIN {X 0,Y 537.772,Z 856.514,A -85,B 0,C 180,E1 21739.696,E2 21739.696} C_VEL
LIN {X 0,Y 534.769,Z 878.539,A -85,B 0,C 180,E1 21738.897,E2 21738.897} C_VEL
LIN {X 0,Y 530.756,Z 904.576,A -85,B 0,C 180,E1 21737.764,E2 21737.764} C_VEL
LIN {X 0,Y 526.74,Z 927.69,A -85,B 0,C 180,E1 21736.56,E2 21736.56} C_VEL
LIN {X 0,Y 522.232,Z 951.849,A -85,B 0,C 180,E1 21735.107,E2 21735.107} C_VEL
LIN {X 0,Y 517.465,Z 975.139,A -85,B 0,C 180,E1 21733.465,E2 21733.465} C_VEL
LIN {X 0,Y 516.685,Z 978.933,A -85,B 0,C 180,E1 21733.18,E2 21733.18} C_VEL
LIN {X 0,Y 514.59,Z 985.361,A -85,B 0,C 180,E1 21732.753,E2 21732.753} C_VEL
LIN {X 0,Y 506.253,Z 1001.703,A -85,B 0,C 180,E1 21731.813,E2 21731.813} C_VEL
LIN {X 0,Y 504.074,Z 1007.734,A -85,B 0,C 180,E1 21731.331,E2 21731.331} C_VEL
LIN {X 0,Y 499.102,Z 1029.301,A -85,B 0,C 180,E1 21729.204,E2 21729.204} C_VEL
LIN {X 0,Y 494.397,Z 1049.525,A -85,B 0,C 180,E1 21726.919,E2 21726.919} C_VEL
LIN {X 0,Y 489.223,Z 1073.28,A -85,B 0,C 180,E1 21723.916,E2 21723.916} C_VEL
LIN {X 0,Y 486.412,Z 1086.584,A -85,B 0,C 180,E1 21722.031,E2 21722.031} C_VEL
LIN {X 0,Y 483.414,Z 1100.81,A -85,B 0,C 180,E1 21719.764,E2 21719.764} C_VEL
LIN {X 0,Y 480.344,Z 1115.482,A -85,B 0,C 180,E1 21717.009,E2 21717.009} C_VEL
LIN {X 0,Y 478.213,Z 1126.033,A -85,B 0,C 180,E1 21714.721,E2 21714.721} C_VEL
LIN {X 0,Y 476.477,Z 1135.201,A -85,B 0,C 180,E1 21712.454,E2 21712.454} C_VEL
LIN {X 0,Y 475.006,Z 1143.544,A -85,B 0,C 180,E1 21710.068,E2 21710.068} C_VEL
LIN {X 0,Y 473.798,Z 1151.439,A -85,B 0,C 180,E1 21707.439,E2 21707.439} C_VEL
LIN {X 0,Y 472.777,Z 1159.716,A -85,B 0,C 180,E1 21704.078,E2 21704.078} C_VEL
LIN {X 0,Y 472.245,Z 1165.609,A -85,B 0,C 180,E1 21700.987,E2 21700.987} C_VEL
LIN {X 0,Y 472.033,Z 1169.6,A -85,B 0,C 180,E1 21698.283,E2 21698.283} C_VEL
LIN {X 0,Y 471.94,Z 1172.367,A -85,B 0,C 180,E1 21695.716,E2 21695.716} C_VEL
LIN {X 0,Y 471.912,Z 1174.172,A -85,B 0,C 180,E1 21693.038,E2 21693.038} C_VEL
LIN {X 0,Y 471.895,Z 1174.882,A -85,B 0,C 180,E1 21690.487,E2 21690.487} C_VEL
LIN {X 0,Y 471.91,Z 1174.55,A -85,B 0,C 180,E1 21687.816,E2 21687.816} C_VEL
LIN {X 0,Y 471.92,Z 1173.221,A -85,B 0,C 180,E1 21685.262,E2 21685.262} C_VEL
LIN {X 0,Y 471.988,Z 1170.74,A -85,B 0,C 180,E1 21682.577,E2 21682.577} C_VEL
LIN {X 0,Y 472.142,Z 1167.31,A -85,B 0,C 180,E1 21679.987,E2 21679.987} C_VEL
LIN {X 0,Y 472.479,Z 1162.628,A -85,B 0,C 180,E1 21677.287,E2 21677.287} C_VEL
LIN {X 0,Y 473.068,Z 1157.039,A -85,B 0,C 180,E1 21674.682,E2 21674.682} C_VEL
LIN {X 0,Y 473.905,Z 1150.634,A -85,B 0,C 180,E1 21672.187,E2 21672.187} C_VEL
LIN {X 0,Y 475.022,Z 1143.431,A -85,B 0,C 180,E1 21669.807,E2 21669.807} C_VEL
LIN {X 0,Y 476.514,Z 1135.033,A -85,B 0,C 180,E1 21667.41,E2 21667.41} C_VEL
LIN {X 0,Y 478.35,Z 1125.362,A -85,B 0,C 180,E1 21665.026,E2 21665.026} C_VEL
LIN {X 0,Y 481.014,Z 1112.321,A -85,B 0,C 180,E1 21662.251,E2 21662.251} C_VEL
LIN {X 0,Y 483.778,Z 1099.051,A -85,B 0,C 180,E1 21659.854,E2 21659.854} C_VEL
LIN {X 0,Y 486.658,Z 1085.49,A -85,B 0,C 180,E1 21657.713,E2 21657.713} C_VEL
LIN {X 0,Y 489.895,Z 1070.148,A -85,B 0,C 180,E1 21655.575,E2 21655.575} C_VEL
LIN {X 0,Y 494.845,Z 1047.585,A -85,B 0,C 180,E1 21652.762,E2 21652.762} C_VEL
LIN {X 0,Y 499.761,Z 1026.526,A -85,B 0,C 180,E1 21650.417,E2 21650.417} C_VEL
LIN {X 0,Y 504.358,Z 1006.462,A -85,B 0,C 180,E1 21648.462,E2 21648.462} C_VEL
LIN {X 0,Y 508.912,Z 986.354,A -85,B 0,C 180,E1 21646.712,E2 21646.712} C_VEL
LIN {X 0,Y 514.001,Z 962.688,A -85,B 0,C 180,E1 21644.923,E2 21644.923} C_VEL
LIN {X 0,Y 518.341,Z 941.482,A -85,B 0,C 180,E1 21643.524,E2 21643.524} C_VEL
LIN {X 0,Y 523.199,Z 915.669,A -85,B 0,C 180,E1 21642.061,E2 21642.061} C_VEL
LIN {X 0,Y 526.914,Z 893.878,A -85,B 0,C 180,E1 21641.014,E2 21641.014} C_VEL
LIN {X 0,Y 530.841,Z 868.274,A -85,B 0,C 180,E1 21639.97,E2 21639.97} C_VEL
LIN {X 0,Y 534.069,Z 843.001,A -85,B 0,C 180,E1 21639.148,E2 21639.148} C_VEL
LIN {X 0,Y 536.749,Z 818.208,A -85,B 0,C 180,E1 21638.5,E2 21638.5} C_VEL
LIN {X 0,Y 548.241,Z 697.96,A -85,B 0,C 180,E1 21636.002,E2 21636.002} C_VEL
LIN {X 0,Y 557.028,Z 598.871,A -85,B 0,C 180,E1 21634.142,E2 21634.142} C_VEL
LIN {X 0,Y 563.352,Z 513.758,A -85,B 0,C 180,E1 21632.683,E2 21632.683} C_VEL
LIN {X 0,Y 566.177,Z 466.9,A -85,B 0,C 180,E1 21631.933,E2 21631.933} C_VEL
LIN {X 0,Y 555.558,Z 456.954,A -85,B 0,C 180,E1 21629.844,E2 21629.844} C_VEL
LIN {X 0,Y 546.35,Z 449.219,A -85,B 0,C 180,E1 21627.879,E2 21627.879} C_VEL
LIN {X 0,Y 538.308,Z 442.736,A -85,B 0,C 180,E1 21626,E2 21626} C_VEL
LIN {X 0,Y 532.142,Z 438.13,A -85,B 0,C 180,E1 21624.417,E2 21624.417} C_VEL
LIN {X 0,Y 531.444,Z 436.384,A -85,B 0,C 180,E1 21623.273,E2 21623.273} C_VEL
LIN {X 0,Y 529.425,Z 431.917,A -85,B 0,C 180,E1 21618.956,E2 21618.956} C_VEL
LIN {X 0,Y 528.343,Z 430.787,A -85,B 0,C 180,E1 21614.466,E2 21614.466} C_VEL
LIN {X 0,Y 529.069,Z 431.577,A -85,B 0,C 180,E1 21610.343,E2 21610.343} C_VEL
LIN {X 0,Y 529.802,Z 432.595,A -85,B 0,C 180,E1 21608.575,E2 21608.575} C_VEL
LIN {X 0,Y 532.186,Z 437.442,A -85,B 0,C 180,E1 21604.31,E2 21604.31} C_VEL
LIN {X 0,Y 534.557,Z 442.353,A -85,B 0,C 180,E1 21601.393,E2 21601.393} C_VEL
LIN {X 0,Y 536.948,Z 447.235,A -85,B 0,C 180,E1 21599.04,E2 21599.04} C_VEL
LIN {X 0,Y 539.292,Z 452.153,A -85,B 0,C 180,E1 21597.024,E2 21597.024} C_VEL
LIN {X 0,Y 542.578,Z 458.8,A -85,B 0,C 180,E1 21594.607,E2 21594.607} C_VEL
LIN {X 0,Y 546.755,Z 468.033,A -85,B 0,C 180,E1 21591.799,E2 21591.799} C_VEL
LIN {X 0,Y 551.561,Z 479.048,A -85,B 0,C 180,E1 21588.921,E2 21588.921} C_VEL
LIN {X 0,Y 555.333,Z 488.31,A -85,B 0,C 180,E1 21586.808,E2 21586.808} C_VEL
LIN {X 0,Y 548.059,Z 521.665,A -85,B 0,C 180,E1 21583.791,E2 21583.791} C_VEL
LIN {X 0,Y 540.156,Z 560.423,A -85,B 0,C 180,E1 21580.421,E2 21580.421} C_VEL
LIN {X 0,Y 532.85,Z 598.781,A -85,B 0,C 180,E1 21577.195,E2 21577.195} C_VEL
LIN {X 0,Y 529.161,Z 623.323,A -85,B 0,C 180,E1 21575.078,E2 21575.078} C_VEL
LIN {X 0,Y 528.044,Z 643.506,A -85,B 0,C 180,E1 21573.146,E2 21573.146} C_VEL
LIN {X 0,Y 528.965,Z 661.144,A -85,B 0,C 180,E1 21571.289,E2 21571.289} C_VEL
LIN {X 0,Y 531.879,Z 677.83,A -85,B 0,C 180,E1 21569.372,E2 21569.372} C_VEL
LIN {X 0,Y 533.354,Z 682.822,A -85,B 0,C 180,E1 21568.809,E2 21568.809} C_VEL
LIN {X 0,Y 539.041,Z 695.138,A -85,B 0,C 180,E1 21567.536,E2 21567.536} C_VEL
LIN {X 0,Y 549.148,Z 712.308,A -85,B 0,C 180,E1 21565.541,E2 21565.541} C_VEL
LIN {X 0,Y 558.657,Z 724.684,A -85,B 0,C 180,E1 21563.893,E2 21563.893} C_VEL
LIN {X 0,Y 558.896,Z 725.409,A -85,B 0,C 180,E1 21563.844,E2 21563.844} C_VEL
LIN {X 0,Y 554.746,Z 751.007,A -85,B 0,C 180,E1 21563.895,E2 21563.895} C_VEL
LIN {X 0,Y 552.282,Z 772.845,A -85,B 0,C 180,E1 21563.769,E2 21563.769} C_VEL
LIN {X 0,Y 549.469,Z 808.562,A -85,B 0,C 180,E1 21563.16,E2 21563.16} C_VEL
LIN {X 0,Y 545.256,Z 845.823,A -85,B 0,C 180,E1 21562.375,E2 21562.375} C_VEL
LIN {X 0,Y 541.005,Z 877.304,A -85,B 0,C 180,E1 21561.528,E2 21561.528} C_VEL
LIN {X 0,Y 536.493,Z 907.922,A -85,B 0,C 180,E1 21560.494,E2 21560.494} C_VEL
LIN {X 0,Y 531.755,Z 937.668,A -85,B 0,C 180,E1 21559.266,E2 21559.266} C_VEL
LIN {X 0,Y 526.751,Z 966.659,A -85,B 0,C 180,E1 21557.835,E2 21557.835} C_VEL
LIN {X 0,Y 521.725,Z 993.758,A -85,B 0,C 180,E1 21556.26,E2 21556.26} C_VEL
LIN {X 0,Y 516.701,Z 1019.06,A -85,B 0,C 180,E1 21554.544,E2 21554.544} C_VEL
LIN {X 0,Y 512.283,Z 1039.461,A -85,B 0,C 180,E1 21552.934,E2 21552.934} C_VEL
LIN {X 0,Y 507.581,Z 1058.977,A -85,B 0,C 180,E1 21551.141,E2 21551.141} C_VEL
LIN {X 0,Y 502.852,Z 1077.05,A -85,B 0,C 180,E1 21549.219,E2 21549.219} C_VEL
LIN {X 0,Y 498.161,Z 1093.713,A -85,B 0,C 180,E1 21547.166,E2 21547.166} C_VEL
LIN {X 0,Y 493.554,Z 1108.849,A -85,B 0,C 180,E1 21544.98,E2 21544.98} C_VEL
LIN {X 0,Y 489.111,Z 1122.405,A -85,B 0,C 180,E1 21542.661,E2 21542.661} C_VEL
LIN {X 0,Y 484.113,Z 1137.819,A -85,B 0,C 180,E1 21539.577,E2 21539.577} C_VEL
LIN {X 0,Y 479.66,Z 1153.436,A -85,B 0,C 180,E1 21535.959,E2 21535.959} C_VEL
LIN {X 0,Y 476.66,Z 1165.987,A -85,B 0,C 180,E1 21532.572,E2 21532.572} C_VEL
LIN {X 0,Y 474.515,Z 1177.172,A -85,B 0,C 180,E1 21529.061,E2 21529.061} C_VEL
LIN {X 0,Y 473.23,Z 1185.803,A -85,B 0,C 180,E1 21525.815,E2 21525.815} C_VEL
LIN {X 0,Y 472.465,Z 1192.835,A -85,B 0,C 180,E1 21522.589,E2 21522.589} C_VEL
LIN {X 0,Y 472.107,Z 1198.097,A -85,B 0,C 180,E1 21519.507,E2 21519.507} C_VEL
LIN {X 0,Y 471.958,Z 1201.767,A -85,B 0,C 180,E1 21516.445,E2 21516.445} C_VEL
LIN {X 0,Y 471.916,Z 1204.078,A -85,B 0,C 180,E1 21513.4,E2 21513.4} C_VEL
LIN {X 0,Y 471.896,Z 1204.916,A -85,B 0,C 180,E1 21510.606,E2 21510.606} C_VEL
LIN {X 0,Y 471.909,Z 1204.499,A -85,B 0,C 180,E1 21507.57,E2 21507.57} C_VEL
LIN {X 0,Y 471.934,Z 1202.78,A -85,B 0,C 180,E1 21504.65,E2 21504.65} C_VEL
LIN {X 0,Y 472.035,Z 1199.529,A -85,B 0,C 180,E1 21501.584,E2 21501.584} C_VEL
LIN {X 0,Y 472.299,Z 1194.923,A -85,B 0,C 180,E1 21498.52,E2 21498.52} C_VEL
LIN {X 0,Y 472.889,Z 1188.702,A -85,B 0,C 180,E1 21495.425,E2 21495.425} C_VEL
LIN {X 0,Y 473.989,Z 1180.325,A -85,B 0,C 180,E1 21492.061,E2 21492.061} C_VEL
LIN {X 0,Y 475.711,Z 1170.584,A -85,B 0,C 180,E1 21488.805,E2 21488.805} C_VEL
LIN {X 0,Y 478.66,Z 1157.33,A -85,B 0,C 180,E1 21485.04,E2 21485.04} C_VEL
LIN {X 0,Y 482.742,Z 1142.344,A -85,B 0,C 180,E1 21481.414,E2 21481.414} C_VEL
LIN {X 0,Y 487.596,Z 1126.987,A -85,B 0,C 180,E1 21478.195,E2 21478.195} C_VEL
LIN {X 0,Y 492.344,Z 1112.644,A -85,B 0,C 180,E1 21475.625,E2 21475.625} C_VEL
LIN {X 0,Y 496.897,Z 1097.875,A -85,B 0,C 180,E1 21473.408,E2 21473.408} C_VEL
LIN {X 0,Y 501.725,Z 1081.141,A -85,B 0,C 180,E1 21471.26,E2 21471.26} C_VEL
LIN {X 0,Y 506.514,Z 1063.32,A -85,B 0,C 180,E1 21469.292,E2 21469.292} C_VEL
LIN {X 0,Y 511.359,Z 1043.64,A -85,B 0,C 180,E1 21467.424,E2 21467.424} C_VEL
LIN {X 0,Y 515.894,Z 1023.042,A -85,B 0,C 180,E1 21465.753,E2 21465.753} C_VEL
LIN {X 0,Y 521.36,Z 995.454,A -85,B 0,C 180,E1 21463.853,E2 21463.853} C_VEL
LIN {X 0,Y 526.175,Z 969.795,A -85,B 0,C 180,E1 21462.334,E2 21462.334} C_VEL
LIN {X 0,Y 531.236,Z 940.737,A -85,B 0,C 180,E1 21460.875,E2 21460.875} C_VEL
LIN {X 0,Y 536.05,Z 910.628,A -85,B 0,C 180,E1 21459.612,E2 21459.612} C_VEL
LIN {X 0,Y 540.683,Z 879.343,A -85,B 0,C 180,E1 21458.537,E2 21458.537} C_VEL
LIN {X 0,Y 545.107,Z 846.879,A -85,B 0,C 180,E1 21457.651,E2 21457.651} C_VEL
LIN {X 0,Y 549.157,Z 811.615,A -85,B 0,C 180,E1 21456.901,E2 21456.901} C_VEL
LIN {X 0,Y 552.158,Z 772.45,A -85,B 0,C 180,E1 21456.211,E2 21456.211} C_VEL
LIN {X 0,Y 556.384,Z 694.467,A -85,B 0,C 180,E1 21455.109,E2 21455.109} C_VEL
LIN {X 0,Y 561.342,Z 650.286,A -85,B 0,C 180,E1 21454.361,E2 21454.361} C_VEL
LIN {X 0,Y 565.705,Z 613.042,A -85,B 0,C 180,E1 21453.757,E2 21453.757} C_VEL
LIN {X 0,Y 567.272,Z 599.802,A -85,B 0,C 180,E1 21453.545,E2 21453.545} C_VEL
LIN {X 0,Y 571.065,Z 566.73,A -85,B 0,C 180,E1 21452.997,E2 21452.997} C_VEL
LIN {X 0,Y 574.237,Z 542.964,A -85,B 0,C 180,E1 21452.668,E2 21452.668} C_VEL
LIN {X 0,Y 577.566,Z 513.263,A -85,B 0,C 180,E1 21452.165,E2 21452.165} C_VEL
LIN {X 0,Y 581.237,Z 486.641,A -85,B 0,C 180,E1 21451.815,E2 21451.815} C_VEL
LIN {X 0,Y 571.013,Z 469.59,A -85,B 0,C 180,E1 21449.649,E2 21449.649} C_VEL
LIN {X 0,Y 560.918,Z 453.731,A -85,B 0,C 180,E1 21447.324,E2 21447.324} C_VEL
LIN {X 0,Y 552.011,Z 440.518,A -85,B 0,C 180,E1 21445.079,E2 21445.079} C_VEL
LIN {X 0,Y 543.711,Z 428.844,A -85,B 0,C 180,E1 21442.775,E2 21442.775} C_VEL
LIN {X 0,Y 537.504,Z 420.293,A -85,B 0,C 180,E1 21440.869,E2 21440.869} C_VEL
LIN {X 0,Y 532.742,Z 414.144,A -85,B 0,C 180,E1 21439.289,E2 21439.289} C_VEL
LIN {X 0,Y 531.476,Z 412.738,A -85,B 0,C 180,E1 21438.858,E2 21438.858} C_VEL
LIN {X 0,Y 530.175,Z 415.801,A -85,B 0,C 180,E1 21438.665,E2 21438.665} C_VEL
LIN {X 0,Y 525.477,Z 428.828,A -85,B 0,C 180,E1 21438.062,E2 21438.062} C_VEL
LIN {X 0,Y 521.485,Z 438.152,A -85,B 0,C 180,E1 21437.419,E2 21437.419} C_VEL
LIN {X 0,Y 515.976,Z 453.873,A -85,B 0,C 180,E1 21436.667,E2 21436.667} C_VEL
LIN {X 0,Y 512.395,Z 462.478,A -85,B 0,C 180,E1 21436.044,E2 21436.044} C_VEL
LIN {X 0,Y 511.456,Z 465.069,A -85,B 0,C 180,E1 21435.898,E2 21435.898} C_VEL
LIN {X 0,Y 507.241,Z 477.683,A -85,B 0,C 180,E1 21435.294,E2 21435.294} C_VEL
LIN {X 0,Y 504,Z 485.862,A -85,B 0,C 180,E1 21434.696,E2 21434.696} C_VEL
LIN {X 0,Y 503.003,Z 488.253,A -85,B 0,C 180,E1 21434.497,E2 21434.497} C_VEL
LIN {X 0,Y 498.859,Z 501.294,A -85,B 0,C 180,E1 21433.88,E2 21433.88} C_VEL
LIN {X 0,Y 495.816,Z 509.469,A -85,B 0,C 180,E1 21433.291,E2 21433.291} C_VEL
LIN {X 0,Y 494.554,Z 512.509,A -85,B 0,C 180,E1 21433.008,E2 21433.008} C_VEL
LIN {X 0,Y 490.514,Z 525.88,A -85,B 0,C 180,E1 21432.382,E2 21432.382} C_VEL
LIN {X 0,Y 487.74,Z 533.819,A -85,B 0,C 180,E1 21431.815,E2 21431.815} C_VEL
LIN {X 0,Y 486.462,Z 537.135,A -85,B 0,C 180,E1 21431.448,E2 21431.448} C_VEL
LIN {X 0,Y 485.373,Z 612.907,A -85,B 0,C 180,E1 21428.291,E2 21428.291} C_VEL
LIN {X 0,Y 484.057,Z 687.234,A -85,B 0,C 180,E1 21425.126,E2 21425.126} C_VEL
LIN {X 0,Y 482.365,Z 767.039,A -85,B 0,C 180,E1 21421.663,E2 21421.663} C_VEL
LIN {X 0,Y 480.587,Z 847.563,A -85,B 0,C 180,E1 21418.092,E2 21418.092} C_VEL
LIN {X 0,Y 478.793,Z 872.877,A -85,B 0,C 180,E1 21417.037,E2 21417.037} C_VEL
LIN {X 0,Y 477.361,Z 974.876,A -85,B 0,C 180,E1 21415.286,E2 21415.286} C_VEL
LIN {X 0,Y 477.507,Z 992.008,A -85,B 0,C 180,E1 21414.921,E2 21414.921} C_VEL
LIN {X 0,Y 477.477,Z 1006.156,A -85,B 0,C 180,E1 21414.412,E2 21414.412} C_VEL
LIN {X 0,Y 477.297,Z 1018.075,A -85,B 0,C 180,E1 21413.806,E2 21413.806} C_VEL
LIN {X 0,Y 477.043,Z 1028.365,A -85,B 0,C 180,E1 21413.138,E2 21413.138} C_VEL
LIN {X 0,Y 476.714,Z 1038.887,A -85,B 0,C 180,E1 21412.285,E2 21412.285} C_VEL
LIN {X 0,Y 476.239,Z 1050.277,A -85,B 0,C 180,E1 21411.123,E2 21411.123} C_VEL
LIN {X 0,Y 475.765,Z 1059.128,A -85,B 0,C 180,E1 21409.954,E2 21409.954} C_VEL
LIN {X 0,Y 475.369,Z 1065.973,A -85,B 0,C 180,E1 21408.842,E2 21408.842} C_VEL
LIN {X 0,Y 474.989,Z 1071.994,A -85,B 0,C 180,E1 21407.626,E2 21407.626} C_VEL
LIN {X 0,Y 474.662,Z 1076.909,A -85,B 0,C 180,E1 21406.353,E2 21406.353} C_VEL
LIN {X 0,Y 474.374,Z 1081.18,A -85,B 0,C 180,E1 21404.849,E2 21404.849} C_VEL
LIN {X 0,Y 474.13,Z 1084.108,A -85,B 0,C 180,E1 21403.08,E2 21403.08} C_VEL
LIN {X 0,Y 474.024,Z 1085.04,A -85,B 0,C 180,E1 21401.664,E2 21401.664} C_VEL
LIN {X 0,Y 473.985,Z 1084.768,A -85,B 0,C 180,E1 21400.274,E2 21400.274} C_VEL
LIN {X 0,Y 474.01,Z 1083.22,A -85,B 0,C 180,E1 21398.809,E2 21398.809} C_VEL
LIN {X 0,Y 474.173,Z 1079.62,A -85,B 0,C 180,E1 21397.039,E2 21397.039} C_VEL
LIN {X 0,Y 474.398,Z 1074.527,A -85,B 0,C 180,E1 21395.467,E2 21395.467} C_VEL
LIN {X 0,Y 474.704,Z 1068.56,A -85,B 0,C 180,E1 21394.082,E2 21394.082} C_VEL
LIN {X 0,Y 475.136,Z 1060.59,A -85,B 0,C 180,E1 21392.633,E2 21392.633} C_VEL
LIN {X 0,Y 475.638,Z 1050.435,A -85,B 0,C 180,E1 21391.223,E2 21391.223} C_VEL
LIN {X 0,Y 476.081,Z 1040.91,A -85,B 0,C 180,E1 21390.16,E2 21390.16} C_VEL
LIN {X 0,Y 476.503,Z 1030.408,A -85,B 0,C 180,E1 21389.202,E2 21389.202} C_VEL
LIN {X 0,Y 476.955,Z 1016.45,A -85,B 0,C 180,E1 21388.21,E2 21388.21} C_VEL
LIN {X 0,Y 477.216,Z 1004.356,A -85,B 0,C 180,E1 21387.562,E2 21387.562} C_VEL
LIN {X 0,Y 477.357,Z 991.972,A -85,B 0,C 180,E1 21387.063,E2 21387.063} C_VEL
LIN {X 0,Y 477.385,Z 976.877,A -85,B 0,C 180,E1 21386.655,E2 21386.655} C_VEL
LIN {X 0,Y 478.18,Z 900.62,A -85,B 0,C 180,E1 21385.391,E2 21385.391} C_VEL
LIN {X 0,Y 479.221,Z 901.632,A -85,B 0,C 180,E1 21385.131,E2 21385.131} C_VEL
LIN {X 0,Y 480.505,Z 901.217,A -85,B 0,C 180,E1 21384.947,E2 21384.947} C_VEL
LIN {X 0,Y 483.043,Z 898.686,A -85,B 0,C 180,E1 21384.723,E2 21384.723} C_VEL
LIN {X 0,Y 486.446,Z 893.296,A -85,B 0,C 180,E1 21384.574,E2 21384.574} C_VEL
LIN {X 0,Y 487.367,Z 891.675,A -85,B 0,C 180,E1 21384.546,E2 21384.546} C_VEL
LIN {X 0,Y 490.58,Z 889.399,A -85,B 0,C 180,E1 21384.2,E2 21384.2} C_VEL
LIN {X 0,Y 494.269,Z 885.016,A -85,B 0,C 180,E1 21383.936,E2 21383.936} C_VEL
LIN {X 0,Y 498.298,Z 878.28,A -85,B 0,C 180,E1 21383.772,E2 21383.772} C_VEL
LIN {X 0,Y 502.367,Z 874.272,A -85,B 0,C 180,E1 21383.408,E2 21383.408} C_VEL
LIN {X 0,Y 506.875,Z 868.733,A -85,B 0,C 180,E1 21383.082,E2 21383.082} C_VEL
LIN {X 0,Y 511.848,Z 864.993,A -85,B 0,C 180,E1 21382.588,E2 21382.588} C_VEL
LIN {X 0,Y 517.773,Z 858.845,A -85,B 0,C 180,E1 21382.113,E2 21382.113} C_VEL
LIN {X 0,Y 523.695,Z 853.925,A -85,B 0,C 180,E1 21381.576,E2 21381.576} C_VEL
LIN {X 0,Y 528.945,Z 848.27,A -85,B 0,C 180,E1 21381.162,E2 21381.162} C_VEL
LIN {X 0,Y 533.897,Z 844.237,A -85,B 0,C 180,E1 21380.725,E2 21380.725} C_VEL
LIN {X 0,Y 530.55,Z 870.173,A -85,B 0,C 180,E1 21379.868,E2 21379.868} C_VEL
LIN {X 0,Y 526.67,Z 895.293,A -85,B 0,C 180,E1 21378.831,E2 21378.831} C_VEL
LIN {X 0,Y 522.469,Z 919.997,A -85,B 0,C 180,E1 21377.623,E2 21377.623} C_VEL
LIN {X 0,Y 518.029,Z 942.975,A -85,B 0,C 180,E1 21376.29,E2 21376.29} C_VEL
LIN {X 0,Y 513.705,Z 964.107,A -85,B 0,C 180,E1 21374.887,E2 21374.887} C_VEL
LIN {X 0,Y 508.458,Z 988.342,A -85,B 0,C 180,E1 21373.031,E2 21373.031} C_VEL
LIN {X 0,Y 504.074,Z 1007.734,A -85,B 0,C 180,E1 21371.331,E2 21371.331} C_VEL
LIN {X 0,Y 501.897,Z 1013.873,A -85,B 0,C 180,E1 21370.836,E2 21370.836} C_VEL
LIN {X 0,Y 492.888,Z 1030.1,A -85,B 0,C 180,E1 21369.642,E2 21369.642} C_VEL
LIN {X 0,Y 491.059,Z 1034.889,A -85,B 0,C 180,E1 21369.161,E2 21369.161} C_VEL
LIN {X 0,Y 486.412,Z 1054.114,A -85,B 0,C 180,E1 21366.889,E2 21366.889} C_VEL
LIN {X 0,Y 481.822,Z 1073.226,A -85,B 0,C 180,E1 21364.316,E2 21364.316} C_VEL
LIN {X 0,Y 477.314,Z 1093.545,A -85,B 0,C 180,E1 21361.274,E2 21361.274} C_VEL
LIN {X 0,Y 474.474,Z 1106.76,A -85,B 0,C 180,E1 21358.994,E2 21358.994} C_VEL
LIN {X 0,Y 472.119,Z 1117.915,A -85,B 0,C 180,E1 21356.816,E2 21356.816} C_VEL
LIN {X 0,Y 470.138,Z 1127.651,A -85,B 0,C 180,E1 21354.637,E2 21354.637} C_VEL
LIN {X 0,Y 468.31,Z 1137.184,A -85,B 0,C 180,E1 21352.206,E2 21352.206} C_VEL
LIN {X 0,Y 466.623,Z 1147.076,A -85,B 0,C 180,E1 21349.27,E2 21349.27} C_VEL
LIN {X 0,Y 465.357,Z 1155.46,A -85,B 0,C 180,E1 21346.167,E2 21346.167} C_VEL
LIN {X 0,Y 464.656,Z 1161.529,A -85,B 0,C 180,E1 21343.44,E2 21343.44} C_VEL
LIN {X 0,Y 464.235,Z 1166.229,A -85,B 0,C 180,E1 21340.802,E2 21340.802} C_VEL
LIN {X 0,Y 464.03,Z 1169.892,A -85,B 0,C 180,E1 21338.178,E2 21338.178} C_VEL
LIN {X 0,Y 463.939,Z 1172.462,A -85,B 0,C 180,E1 21335.691,E2 21335.691} C_VEL
LIN {X 0,Y 463.912,Z 1174.169,A -85,B 0,C 180,E1 21333.09,E2 21333.09} C_VEL
LIN {X 0,Y 463.896,Z 1174.879,A -85,B 0,C 180,E1 21330.495,E2 21330.495} C_VEL
LIN {X 0,Y 463.909,Z 1174.547,A -85,B 0,C 180,E1 21327.778,E2 21327.778} C_VEL
LIN {X 0,Y 463.922,Z 1173.218,A -85,B 0,C 180,E1 21325.18,E2 21325.18} C_VEL
LIN {X 0,Y 463.989,Z 1170.736,A -85,B 0,C 180,E1 21322.448,E2 21322.448} C_VEL
LIN {X 0,Y 464.173,Z 1167.144,A -85,B 0,C 180,E1 21319.702,E2 21319.702} C_VEL
LIN {X 0,Y 464.53,Z 1162.688,A -85,B 0,C 180,E1 21317.066,E2 21317.066} C_VEL
LIN {X 0,Y 465.18,Z 1156.936,A -85,B 0,C 180,E1 21314.358,E2 21314.358} C_VEL
LIN {X 0,Y 466.049,Z 1150.555,A -85,B 0,C 180,E1 21311.877,E2 21311.877} C_VEL
LIN {X 0,Y 467.159,Z 1143.653,A -85,B 0,C 180,E1 21309.583,E2 21309.583} C_VEL
LIN {X 0,Y 468.696,Z 1135.167,A -85,B 0,C 180,E1 21307.155,E2 21307.155} C_VEL
LIN {X 0,Y 470.846,Z 1124.25,A -85,B 0,C 180,E1 21304.465,E2 21304.465} C_VEL
LIN {X 0,Y 473.633,Z 1110.689,A -85,B 0,C 180,E1 21301.643,E2 21301.643} C_VEL
LIN {X 0,Y 476.397,Z 1097.779,A -85,B 0,C 180,E1 21299.337,E2 21299.337} C_VEL
LIN {X 0,Y 479.382,Z 1083.95,A -85,B 0,C 180,E1 21297.162,E2 21297.162} C_VEL
LIN {X 0,Y 484.135,Z 1063.401,A -85,B 0,C 180,E1 21294.236,E2 21294.236} C_VEL
LIN {X 0,Y 488.505,Z 1045.509,A -85,B 0,C 180,E1 21291.971,E2 21291.971} C_VEL
LIN {X 0,Y 493.712,Z 1024.18,A -85,B 0,C 180,E1 21289.596,E2 21289.596} C_VEL
LIN {X 0,Y 498.234,Z 1005.463,A -85,B 0,C 180,E1 21287.758,E2 21287.758} C_VEL
LIN {X 0,Y 503.685,Z 982.267,A -85,B 0,C 180,E1 21285.753,E2 21285.753} C_VEL
LIN {X 0,Y 508.33,Z 961.504,A -85,B 0,C 180,E1 21284.198,E2 21284.198} C_VEL
LIN {X 0,Y 513.348,Z 937.914,A -85,B 0,C 180,E1 21282.647,E2 21282.647} C_VEL
LIN {X 0,Y 517.905,Z 914.026,A -85,B 0,C 180,E1 21281.322,E2 21281.322} C_VEL
LIN {X 0,Y 521.945,Z 891.125,A -85,B 0,C 180,E1 21280.229,E2 21280.229} C_VEL
LIN {X 0,Y 525.855,Z 865.419,A -85,B 0,C 180,E1 21279.212,E2 21279.212} C_VEL
LIN {X 0,Y 528.881,Z 842.542,A -85,B 0,C 180,E1 21278.475,E2 21278.475} C_VEL
LIN {X 0,Y 531.961,Z 814.327,A -85,B 0,C 180,E1 21277.755,E2 21277.755} C_VEL
LIN {X 0,Y 543.657,Z 697.025,A -85,B 0,C 180,E1 21275.297,E2 21275.297} C_VEL
LIN {X 0,Y 552.443,Z 601.267,A -85,B 0,C 180,E1 21273.489,E2 21273.489} C_VEL
LIN {X 0,Y 558.845,Z 517.978,A -85,B 0,C 180,E1 21272.054,E2 21272.054} C_VEL
LIN {X 0,Y 561.701,Z 472.267,A -85,B 0,C 180,E1 21271.318,E2 21271.318} C_VEL
LIN {X 0,Y 551.269,Z 462.685,A -85,B 0,C 180,E1 21269.204,E2 21269.204} C_VEL
LIN {X 0,Y 544.154,Z 456.599,A -85,B 0,C 180,E1 21267.644,E2 21267.644} C_VEL
LIN {X 0,Y 536.381,Z 450.31,A -85,B 0,C 180,E1 21265.803,E2 21265.803} C_VEL
LIN {X 0,Y 527.282,Z 443.25,A -85,B 0,C 180,E1 21263.349,E2 21263.349} C_VEL
LIN {X 0,Y 525.246,Z 438.742,A -85,B 0,C 180,E1 21258.998,E2 21258.998} C_VEL
LIN {X 0,Y 524.155,Z 437.603,A -85,B 0,C 180,E1 21254.472,E2 21254.472} C_VEL
LIN {X 0,Y 524.845,Z 438.36,A -85,B 0,C 180,E1 21250.427,E2 21250.427} C_VEL
LIN {X 0,Y 525.57,Z 439.355,A -85,B 0,C 180,E1 21248.644,E2 21248.644} C_VEL
LIN {X 0,Y 527.9,Z 444.237,A -85,B 0,C 180,E1 21244.345,E2 21244.345} C_VEL
LIN {X 0,Y 530.165,Z 448.947,A -85,B 0,C 180,E1 21241.513,E2 21241.513} C_VEL
LIN {X 0,Y 532.512,Z 453.836,A -85,B 0,C 180,E1 21239.139,E2 21239.139} C_VEL
LIN {X 0,Y 534.949,Z 459.042,A -85,B 0,C 180,E1 21237,E2 21237} C_VEL
LIN {X 0,Y 538.05,Z 465.457,A -85,B 0,C 180,E1 21234.668,E2 21234.668} C_VEL
LIN {X 0,Y 542.027,Z 474.352,A -85,B 0,C 180,E1 21231.941,E2 21231.941} C_VEL
LIN {X 0,Y 546.755,Z 485.395,A -85,B 0,C 180,E1 21229.036,E2 21229.036} C_VEL
LIN {X 0,Y 549.897,Z 493.517,A -85,B 0,C 180,E1 21227.183,E2 21227.183} C_VEL
LIN {X 0,Y 542.427,Z 526.681,A -85,B 0,C 180,E1 21224.168,E2 21224.168} C_VEL
LIN {X 0,Y 534.369,Z 564.853,A -85,B 0,C 180,E1 21220.829,E2 21220.829} C_VEL
LIN {X 0,Y 526.782,Z 603.341,A -85,B 0,C 180,E1 21217.569,E2 21217.569} C_VEL
LIN {X 0,Y 523.121,Z 627.265,A -85,B 0,C 180,E1 21215.476,E2 21215.476} C_VEL
LIN {X 0,Y 521.934,Z 647.109,A -85,B 0,C 180,E1 21213.55,E2 21213.55} C_VEL
LIN {X 0,Y 522.781,Z 665.246,A -85,B 0,C 180,E1 21211.615,E2 21211.615} C_VEL
LIN {X 0,Y 523.844,Z 672.337,A -85,B 0,C 180,E1 21210.842,E2 21210.842} C_VEL
LIN {X 0,Y 528.231,Z 684.529,A -85,B 0,C 180,E1 21209.689,E2 21209.689} C_VEL
LIN {X 0,Y 535.004,Z 699.958,A -85,B 0,C 180,E1 21208.1,E2 21208.1} C_VEL
LIN {X 0,Y 545.458,Z 718.145,A -85,B 0,C 180,E1 21205.974,E2 21205.974} C_VEL
LIN {X 0,Y 553.516,Z 729.31,A -85,B 0,C 180,E1 21204.525,E2 21204.525} C_VEL
LIN {X 0,Y 550.091,Z 750.701,A -85,B 0,C 180,E1 21204.569,E2 21204.569} C_VEL
LIN {X 0,Y 547.511,Z 772.674,A -85,B 0,C 180,E1 21204.439,E2 21204.439} C_VEL
LIN {X 0,Y 544.72,Z 806.195,A -85,B 0,C 180,E1 21203.865,E2 21203.865} C_VEL
LIN {X 0,Y 540.413,Z 843.413,A -85,B 0,C 180,E1 21203.082,E2 21203.082} C_VEL
LIN {X 0,Y 535.896,Z 875.811,A -85,B 0,C 180,E1 21202.215,E2 21202.215} C_VEL
LIN {X 0,Y 531.121,Z 906.912,A -85,B 0,C 180,E1 21201.163,E2 21201.163} C_VEL
LIN {X 0,Y 526.183,Z 936.783,A -85,B 0,C 180,E1 21199.929,E2 21199.929} C_VEL
LIN {X 0,Y 521.289,Z 964.488,A -85,B 0,C 180,E1 21198.566,E2 21198.566} C_VEL
LIN {X 0,Y 516.297,Z 990.777,A -85,B 0,C 180,E1 21197.056,E2 21197.056} C_VEL
LIN {X 0,Y 511.051,Z 1016.589,A -85,B 0,C 180,E1 21195.33,E2 21195.33} C_VEL
LIN {X 0,Y 506.446,Z 1037.372,A -85,B 0,C 180,E1 21193.708,E2 21193.708} C_VEL
LIN {X 0,Y 501.555,Z 1057.284,A -85,B 0,C 180,E1 21191.899,E2 21191.899} C_VEL
LIN {X 0,Y 496.335,Z 1076.743,A -85,B 0,C 180,E1 21189.836,E2 21189.836} C_VEL
LIN {X 0,Y 491.486,Z 1093.639,A -85,B 0,C 180,E1 21187.758,E2 21187.758} C_VEL
LIN {X 0,Y 486.51,Z 1109.995,A -85,B 0,C 180,E1 21185.418,E2 21185.418} C_VEL
LIN {X 0,Y 482.017,Z 1124.017,A -85,B 0,C 180,E1 21183.061,E2 21183.061} C_VEL
LIN {X 0,Y 477.782,Z 1136.552,A -85,B 0,C 180,E1 21180.565,E2 21180.565} C_VEL
LIN {X 0,Y 473.121,Z 1151.103,A -85,B 0,C 180,E1 21177.159,E2 21177.159} C_VEL
LIN {X 0,Y 469.327,Z 1165.168,A -85,B 0,C 180,E1 21173.33,E2 21173.33} C_VEL
LIN {X 0,Y 466.917,Z 1176.2,A -85,B 0,C 180,E1 21169.775,E2 21169.775} C_VEL
LIN {X 0,Y 465.345,Z 1185.672,A -85,B 0,C 180,E1 21166.162,E2 21166.162} C_VEL
LIN {X 0,Y 464.51,Z 1192.811,A -85,B 0,C 180,E1 21162.808,E2 21162.808} C_VEL
LIN {X 0,Y 464.112,Z 1198.268,A -85,B 0,C 180,E1 21159.547,E2 21159.547} C_VEL
LIN {X 0,Y 463.961,Z 1201.794,A -85,B 0,C 180,E1 21156.529,E2 21156.529} C_VEL
LIN {X 0,Y 463.917,Z 1204.13,A -85,B 0,C 180,E1 21153.335,E2 21153.335} C_VEL
LIN {X 0,Y 463.896,Z 1204.934,A -85,B 0,C 180,E1 21150.492,E2 21150.492} C_VEL
LIN {X 0,Y 463.91,Z 1204.445,A -85,B 0,C 180,E1 21147.404,E2 21147.404} C_VEL
LIN {X 0,Y 463.937,Z 1202.691,A -85,B 0,C 180,E1 21144.433,E2 21144.433} C_VEL
LIN {X 0,Y 464.053,Z 1199.381,A -85,B 0,C 180,E1 21141.324,E2 21141.324} C_VEL
LIN {X 0,Y 464.354,Z 1194.675,A -85,B 0,C 180,E1 21138.195,E2 21138.195} C_VEL
LIN {X 0,Y 465.033,Z 1188.151,A -85,B 0,C 180,E1 21134.919,E2 21134.919} C_VEL
LIN {X 0,Y 466.272,Z 1179.747,A -85,B 0,C 180,E1 21131.494,E2 21131.494} C_VEL
LIN {X 0,Y 468.365,Z 1169.179,A -85,B 0,C 180,E1 21127.9,E2 21127.9} C_VEL
LIN {X 0,Y 471.457,Z 1156.818,A -85,B 0,C 180,E1 21124.338,E2 21124.338} C_VEL
LIN {X 0,Y 475.751,Z 1142.738,A -85,B 0,C 180,E1 21120.816,E2 21120.816} C_VEL
LIN {X 0,Y 480.248,Z 1129.271,A -85,B 0,C 180,E1 21117.929,E2 21117.929} C_VEL
LIN {X 0,Y 484.778,Z 1115.352,A -85,B 0,C 180,E1 21115.443,E2 21115.443} C_VEL
LIN {X 0,Y 489.601,Z 1099.911,A -85,B 0,C 180,E1 21113.099,E2 21113.099} C_VEL
LIN {X 0,Y 494.773,Z 1082.438,A -85,B 0,C 180,E1 21110.827,E2 21110.827} C_VEL
LIN {X 0,Y 499.837,Z 1064.031,A -85,B 0,C 180,E1 21108.778,E2 21108.778} C_VEL
LIN {X 0,Y 504.822,Z 1044.332,A -85,B 0,C 180,E1 21106.894,E2 21106.894} C_VEL
LIN {X 0,Y 509.688,Z 1023.026,A -85,B 0,C 180,E1 21105.149,E2 21105.149} C_VEL
LIN {X 0,Y 515.394,Z 995.19,A -85,B 0,C 180,E1 21103.223,E2 21103.223} C_VEL
LIN {X 0,Y 520.73,Z 967.408,A -85,B 0,C 180,E1 21101.59,E2 21101.59} C_VEL
LIN {X 0,Y 525.994,Z 937.943,A -85,B 0,C 180,E1 21100.123,E2 21100.123} C_VEL
LIN {X 0,Y 530.998,Z 907.551,A -85,B 0,C 180,E1 21098.863,E2 21098.863} C_VEL
LIN {X 0,Y 535.831,Z 875.943,A -85,B 0,C 180,E1 21097.793,E2 21097.793} C_VEL
LIN {X 0,Y 540.35,Z 843.704,A -85,B 0,C 180,E1 21096.927,E2 21096.927} C_VEL
LIN {X 0,Y 544.514,Z 808.078,A -85,B 0,C 180,E1 21096.173,E2 21096.173} C_VEL
LIN {X 0,Y 547.617,Z 768.494,A -85,B 0,C 180,E1 21095.476,E2 21095.476} C_VEL
LIN {X 0,Y 551.995,Z 690.411,A -85,B 0,C 180,E1 21094.372,E2 21094.372} C_VEL
LIN {X 0,Y 556.499,Z 651.347,A -85,B 0,C 180,E1 21093.717,E2 21093.717} C_VEL
LIN {X 0,Y 560.928,Z 613.976,A -85,B 0,C 180,E1 21093.108,E2 21093.108} C_VEL
LIN {X 0,Y 562.583,Z 600.235,A -85,B 0,C 180,E1 21092.888,E2 21092.888} C_VEL
LIN {X 0,Y 566.491,Z 566.799,A -85,B 0,C 180,E1 21092.335,E2 21092.335} C_VEL
LIN {X 0,Y 569.64,Z 543.457,A -85,B 0,C 180,E1 21092.013,E2 21092.013} C_VEL
LIN {X 0,Y 573.085,Z 513.344,A -85,B 0,C 180,E1 21091.505,E2 21091.505} C_VEL
LIN {X 0,Y 576.209,Z 490.533,A -85,B 0,C 180,E1 21091.197,E2 21091.197} C_VEL
LIN {X 0,Y 565.962,Z 473.354,A -85,B 0,C 180,E1 21088.952,E2 21088.952} C_VEL
LIN {X 0,Y 555.148,Z 456.373,A -85,B 0,C 180,E1 21086.358,E2 21086.358} C_VEL
LIN {X 0,Y 545.473,Z 442.159,A -85,B 0,C 180,E1 21083.783,E2 21083.783} C_VEL
LIN {X 0,Y 538.06,Z 431.748,A -85,B 0,C 180,E1 21081.589,E2 21081.589} C_VEL
LIN {X 0,Y 533.942,Z 426.261,A -85,B 0,C 180,E1 21080.27,E2 21080.27} C_VEL
LIN {X 0,Y 531.103,Z 422.306,A -85,B 0,C 180,E1 21079.294,E2 21079.294} C_VEL
LIN {X 0,Y 526.322,Z 434.959,A -85,B 0,C 180,E1 21078.67,E2 21078.67} C_VEL
LIN {X 0,Y 522.413,Z 444.073,A -85,B 0,C 180,E1 21078.063,E2 21078.063} C_VEL
LIN {X 0,Y 517.799,Z 457.152,A -85,B 0,C 180,E1 21077.457,E2 21077.457} C_VEL
LIN {X 0,Y 513.837,Z 466.668,A -85,B 0,C 180,E1 21076.802,E2 21076.802} C_VEL
LIN {X 0,Y 512.721,Z 469.736,A -85,B 0,C 180,E1 21076.637,E2 21076.637} C_VEL
LIN {X 0,Y 508.335,Z 482.461,A -85,B 0,C 180,E1 21076.014,E2 21076.014} C_VEL
LIN {X 0,Y 504.813,Z 491.097,A -85,B 0,C 180,E1 21075.377,E2 21075.377} C_VEL
LIN {X 0,Y 503.866,Z 493.727,A -85,B 0,C 180,E1 21075.222,E2 21075.222} C_VEL
LIN {X 0,Y 499.606,Z 506.628,A -85,B 0,C 180,E1 21074.584,E2 21074.584} C_VEL
LIN {X 0,Y 496.363,Z 514.985,A -85,B 0,C 180,E1 21073.959,E2 21073.959} C_VEL
LIN {X 0,Y 495.436,Z 517.403,A -85,B 0,C 180,E1 21073.777,E2 21073.777} C_VEL
LIN {X 0,Y 491.236,Z 530.835,A -85,B 0,C 180,E1 21073.125,E2 21073.125} C_VEL
LIN {X 0,Y 488.253,Z 539.057,A -85,B 0,C 180,E1 21072.522,E2 21072.522} C_VEL
LIN {X 0,Y 487.016,Z 542.163,A -85,B 0,C 180,E1 21072.236,E2 21072.236} C_VEL
LIN {X 0,Y 483.055,Z 555.632,A -85,B 0,C 180,E1 21071.606,E2 21071.606} C_VEL
LIN {X 0,Y 480.164,Z 564.248,A -85,B 0,C 180,E1 21070.999,E2 21070.999} C_VEL
LIN {X 0,Y 478.849,Z 567.659,A -85,B 0,C 180,E1 21070.619,E2 21070.619} C_VEL
LIN {X 0,Y 477.46,Z 651.301,A -85,B 0,C 180,E1 21067.067,E2 21067.067} C_VEL
LIN {X 0,Y 475.534,Z 739.105,A -85,B 0,C 180,E1 21063.255,E2 21063.255} C_VEL
LIN {X 0,Y 473.73,Z 817.243,A -85,B 0,C 180,E1 21059.788,E2 21059.788} C_VEL
LIN {X 0,Y 472.651,Z 856.058,A -85,B 0,C 180,E1 21058.06,E2 21058.06} C_VEL
LIN {X 0,Y 471.142,Z 874.428,A -85,B 0,C 180,E1 21057.305,E2 21057.305} C_VEL
LIN {X 0,Y 469.622,Z 976.003,A -85,B 0,C 180,E1 21055.512,E2 21055.512} C_VEL
LIN {X 0,Y 469.77,Z 993.043,A -85,B 0,C 180,E1 21055.143,E2 21055.143} C_VEL
LIN {X 0,Y 469.737,Z 1007.271,A -85,B 0,C 180,E1 21054.626,E2 21054.626} C_VEL
LIN {X 0,Y 469.537,Z 1019.626,A -85,B 0,C 180,E1 21053.986,E2 21053.986} C_VEL
LIN {X 0,Y 469.262,Z 1030.371,A -85,B 0,C 180,E1 21053.27,E2 21053.27} C_VEL
LIN {X 0,Y 468.873,Z 1042.167,A -85,B 0,C 180,E1 21052.279,E2 21052.279} C_VEL
LIN {X 0,Y 468.349,Z 1052.947,A -85,B 0,C 180,E1 21051.096,E2 21051.096} C_VEL
LIN {X 0,Y 467.916,Z 1060.748,A -85,B 0,C 180,E1 21050.032,E2 21050.032} C_VEL
LIN {X 0,Y 467.502,Z 1067.518,A -85,B 0,C 180,E1 21048.902,E2 21048.902} C_VEL
LIN {X 0,Y 467.098,Z 1073.574,A -85,B 0,C 180,E1 21047.639,E2 21047.639} C_VEL
LIN {X 0,Y 466.738,Z 1078.738,A -85,B 0,C 180,E1 21046.243,E2 21046.243} C_VEL
LIN {X 0,Y 466.392,Z 1083.245,A -85,B 0,C 180,E1 21044.455,E2 21044.455} C_VEL
LIN {X 0,Y 466.208,Z 1085.311,A -85,B 0,C 180,E1 21043.041,E2 21043.041} C_VEL
LIN {X 0,Y 466.099,Z 1086.167,A -85,B 0,C 180,E1 21041.618,E2 21041.618} C_VEL
LIN {X 0,Y 466.061,Z 1085.817,A -85,B 0,C 180,E1 21040.185,E2 21040.185} C_VEL
LIN {X 0,Y 466.099,Z 1084.061,A -85,B 0,C 180,E1 21038.611,E2 21038.611} C_VEL
LIN {X 0,Y 466.279,Z 1080.023,A -85,B 0,C 180,E1 21036.761,E2 21036.761} C_VEL
LIN {X 0,Y 466.509,Z 1075.208,A -85,B 0,C 180,E1 21035.294,E2 21035.294} C_VEL
LIN {X 0,Y 466.818,Z 1069.434,A -85,B 0,C 180,E1 21033.954,E2 21033.954} C_VEL
LIN {X 0,Y 467.275,Z 1061.317,A -85,B 0,C 180,E1 21032.47,E2 21032.47} C_VEL
LIN {X 0,Y 467.791,Z 1051.144,A -85,B 0,C 180,E1 21031.052,E2 21031.052} C_VEL
LIN {X 0,Y 468.262,Z 1041.388,A -85,B 0,C 180,E1 21029.957,E2 21029.957} C_VEL
LIN {X 0,Y 468.77,Z 1029.052,A -85,B 0,C 180,E1 21028.842,E2 21028.842} C_VEL
LIN {X 0,Y 469.172,Z 1016.005,A -85,B 0,C 180,E1 21027.949,E2 21027.949} C_VEL
LIN {X 0,Y 469.437,Z 1003.978,A -85,B 0,C 180,E1 21027.312,E2 21027.312} C_VEL
LIN {X 0,Y 469.599,Z 989.614,A -85,B 0,C 180,E1 21026.751,E2 21026.751} C_VEL
LIN {X 0,Y 469.563,Z 972.399,A -85,B 0,C 180,E1 21026.358,E2 21026.358} C_VEL
LIN {X 0,Y 470.201,Z 916.136,A -85,B 0,C 180,E1 21025.404,E2 21025.404} C_VEL
LIN {X 0,Y 471.027,Z 917.014,A -85,B 0,C 180,E1 21025.178,E2 21025.178} C_VEL
LIN {X 0,Y 472.243,Z 916.814,A -85,B 0,C 180,E1 21024.985,E2 21024.985} C_VEL
LIN {X 0,Y 474.695,Z 914.763,A -85,B 0,C 180,E1 21024.749,E2 21024.749} C_VEL
LIN {X 0,Y 478.037,Z 910.145,A -85,B 0,C 180,E1 21024.592,E2 21024.592} C_VEL
LIN {X 0,Y 479.217,Z 908.403,A -85,B 0,C 180,E1 21024.546,E2 21024.546} C_VEL
LIN {X 0,Y 482.225,Z 906.397,A -85,B 0,C 180,E1 21024.216,E2 21024.216} C_VEL
LIN {X 0,Y 486.067,Z 902.221,A -85,B 0,C 180,E1 21023.945,E2 21023.945} C_VEL
LIN {X 0,Y 489.404,Z 897.183,A -85,B 0,C 180,E1 21023.806,E2 21023.806} C_VEL
LIN {X 0,Y 493.493,Z 893.522,A -85,B 0,C 180,E1 21023.438,E2 21023.438} C_VEL
LIN {X 0,Y 497.904,Z 887.878,A -85,B 0,C 180,E1 21023.169,E2 21023.169} C_VEL
LIN {X 0,Y 500.803,Z 883.237,A -85,B 0,C 180,E1 21023.06,E2 21023.06} C_VEL
LIN {X 0,Y 505.636,Z 878.21,A -85,B 0,C 180,E1 21022.692,E2 21022.692} C_VEL
LIN {X 0,Y 508.741,Z 874.645,A -85,B 0,C 180,E1 21022.462,E2 21022.462} C_VEL
LIN {X 0,Y 514.27,Z 870.21,A -85,B 0,C 180,E1 21021.95,E2 21021.95} C_VEL
LIN {X 0,Y 519.408,Z 864.941,A -85,B 0,C 180,E1 21021.553,E2 21021.553} C_VEL
LIN {X 0,Y 525.891,Z 859.523,A -85,B 0,C 180,E1 21020.998,E2 21020.998} C_VEL
LIN {X 0,Y 526.79,Z 858.742,A -85,B 0,C 180,E1 21020.925,E2 21020.925} C_VEL
